  MoveL 616 to (-197.85, 161.14, -4.14) mm, rotated rx 163.15 ry -25.3 rz 35.32 deg; joints [1.714, -40.378, 129.098, -150.279, 73.685, 65.031, 129.162]
  Set speed (76.2 mm/s)
  MoveL 617 to (-197.85, 161.14, -8.4) mm, rotated rx 163.15 ry -25.3 rz 35.32 deg; joints [1.504, -40.382, 129.115, -150.492, 73.695, 65.043, 129.162]
  MoveL 618 to (-199.6, 161.14, -8.41) mm, rotated rx 163.04 ry -25.23 rz 35.58 deg; joints [1.487, -40.261, 129.125, -150.604, 73.811, 65.026, 128.915]
  MoveL 619 to (-206.05, 161.14, -11.57) mm, rotated rx 162.65 ry -24.96 rz 36.52 deg; joints [1.269, -39.819, 129.168, -151.166, 74.241, 64.973, 128.027]
  MoveL 620 to (-201.08, 161.14, -20.25) mm, rotated rx 162.95 ry -25.17 rz 35.8 deg; joints [0.888, -40.168, 129.175, -151.29, 73.933, 65.037, 128.708]
  MoveL 621 to (-201.08, 157.97, -20.25) mm, rotated rx 162.7 ry -25 rz 36.39 deg; joints [0.848, -40.277, 129.313, -151.506, 73.963, 64.865, 128.153]
  MoveL 622 to (-206.05, 157.97, -11.57) mm, rotated rx 162.4 ry -24.8 rz 37.1 deg; joints [1.229, -39.927, 129.307, -151.385, 74.271, 64.804, 127.476]
  MoveL 623 to (-199.6, 157.97, -8.41) mm, rotated rx 162.79 ry -25.06 rz 36.17 deg; joints [1.449, -40.37, 129.264, -150.819, 73.841, 64.853, 128.359]
  MoveL 624 to (-197.85, 157.97, -8.4) mm, rotated rx 162.9 ry -25.13 rz 35.91 deg; joints [1.466, -40.491, 129.254, -150.707, 73.725, 64.869, 128.605]
  MoveL 625 to (-197.85, 157.97, -4.14) mm, rotated rx 162.9 ry -25.13 rz 35.91 deg; joints [1.676, -40.487, 129.236, -150.493, 73.716, 64.858, 128.605]
  Set speed (38.1 mm/s)
  MoveL 626 to (-197.89, 157.97, -3.98) mm, rotated rx 162.9 ry -25.13 rz 35.92 deg; joints [1.684, -40.484, 129.236, -150.488, 73.718, 64.857, 128.599]
  MoveL 627 to (-198.05, 157.65, -3.7) mm, rotated rx 162.87 ry -25.11 rz 36 deg; joints [1.692, -40.484, 129.25, -150.506, 73.731, 64.838, 128.521]
  Set speed (76.2 mm/s)
  MoveL 628 to (-198.05, 155.11, -3.7) mm, rotated rx 162.66 ry -24.98 rz 36.48 deg; joints [1.661, -40.571, 129.362, -150.683, 73.756, 64.699, 128.068]
  Set speed (38.1 mm/s)
  MoveL 629 to (-197.89, 154.79, -3.98) mm, rotated rx 162.65 ry -24.97 rz 36.51 deg; joints [1.644, -40.593, 129.376, -150.709, 73.749, 64.684, 128.033]
  MoveL 630 to (-197.85, 154.79, -4.14) mm, rotated rx 162.65 ry -24.97 rz 36.51 deg; joints [1.637, -40.596, 129.377, -150.714, 73.747, 64.685, 128.039]
  Set speed (76.2 mm/s)
  MoveL 631 to (-197.85, 154.79, -8.4) mm, rotated rx 162.65 ry -24.97 rz 36.51 deg; joints [1.426, -40.6, 129.394, -150.928, 73.756, 64.695, 128.039]
  MoveL 632 to (-199.6, 154.79, -8.41) mm, rotated rx 162.54 ry -24.89 rz 36.76 deg; joints [1.409, -40.479, 129.404, -151.041, 73.873, 64.68, 127.794]
  MoveL 633 to (-206.05, 154.79, -11.57) mm, rotated rx 162.16 ry -24.63 rz 37.69 deg; joints [1.188, -40.035, 129.447, -151.609, 74.302, 64.635, 126.915]
  MoveL 634 to (-201.08, 154.79, -20.25) mm, rotated rx 162.45 ry -24.83 rz 36.98 deg; joints [0.808, -40.386, 129.453, -151.729, 73.993, 64.693, 127.59]
  MoveL 635 to (-201.08, 151.62, -20.25) mm, rotated rx 162.2 ry -24.66 rz 37.58 deg; joints [0.765, -40.493, 129.594, -151.959, 74.025, 64.521, 127.017]
  MoveL 636 to (-206.05, 151.62, -11.57) mm, rotated rx 161.91 ry -24.45 rz 38.28 deg; joints [1.146, -40.142, 129.589, -151.84, 74.333, 64.466, 126.347]
  MoveL 637 to (-199.6, 151.62, -8.41) mm, rotated rx 162.29 ry -24.72 rz 37.37 deg; joints [1.367, -40.587, 129.546, -151.27, 73.905, 64.508, 127.221]
  MoveL 638 to (-197.85, 151.62, -8.4) mm, rotated rx 162.4 ry -24.79 rz 37.11 deg; joints [1.385, -40.708, 129.536, -151.156, 73.789, 64.522, 127.465]
  MoveL 639 to (-197.85, 151.62, -4.14) mm, rotated rx 162.4 ry -24.79 rz 37.11 deg; joints [1.596, -40.704, 129.519, -150.942, 73.779, 64.512, 127.465]
  Set speed (38.1 mm/s)
  MoveL 640 to (-197.89, 151.62, -3.98) mm, rotated rx 162.39 ry -24.79 rz 37.12 deg; joints [1.604, -40.701, 129.518, -150.937, 73.782, 64.511, 127.459]
  MoveL 641 to (-198.05, 151.3, -3.7) mm, rotated rx 162.36 ry -24.77 rz 37.2 deg; joints [1.612, -40.701, 129.533, -150.956, 73.795, 64.492, 127.378]
  Set speed (76.2 mm/s)
  MoveL 642 to (-198.05, 148.76, -3.7) mm, rotated rx 162.15 ry -24.63 rz 37.69 deg; joints [1.578, -40.786, 129.648, -151.144, 73.821, 64.354, 126.912]
  Set speed (38.1 mm/s)
  MoveL 643 to (-197.89, 148.44, -3.98) mm, rotated rx 162.14 ry -24.62 rz 37.73 deg; joints [1.562, -40.808, 129.663, -151.171, 73.815, 64.339, 126.875]
  MoveL 644 to (-197.85, 148.44, -4.14) mm, rotated rx 162.14 ry -24.62 rz 37.72 deg; joints [1.554, -40.812, 129.663, -151.176, 73.812, 64.339, 126.881]
  Set speed (76.2 mm/s)
  MoveL 645 to (-197.85, 148.44, -8.4) mm, rotated rx 162.14 ry -24.62 rz 37.72 deg; joints [1.343, -40.815, 129.68, -151.391, 73.822, 64.35, 126.881]
  MoveL 646 to (-199.6, 148.44, -8.41) mm, rotated rx 162.04 ry -24.54 rz 37.98 deg; joints [1.325, -40.694, 129.69, -151.505, 73.937, 64.337, 126.639]
  MoveL 647 to (-206.05, 148.44, -11.57) mm, rotated rx 161.66 ry -24.27 rz 38.88 deg; joints [1.102, -40.248, 129.733, -152.077, 74.366, 64.298, 125.77]
  MoveL 648 to (-201.08, 148.44, -20.25) mm, rotated rx 161.95 ry -24.48 rz 38.19 deg; joints [0.722, -40.6, 129.738, -152.196, 74.058, 64.349, 126.436]
  MoveL 649 to (-201.08, 145.27, -20.25) mm, rotated rx 161.69 ry -24.3 rz 38.8 deg; joints [0.676, -40.706, 129.883, -152.439, 74.091, 64.178, 125.846]
  MoveL 650 to (-206.05, 145.27, -11.57) mm, rotated rx 161.41 ry -24.09 rz 39.49 deg; joints [1.057, -40.353, 129.879, -152.322, 74.399, 64.131, 125.185]
  MoveL 651 to (-199.6, 145.27, -8.41) mm, rotated rx 161.78 ry -24.36 rz 38.59 deg; joints [1.28, -40.8, 129.836, -151.748, 73.971, 64.166, 126.047]
  MoveL 652 to (-197.85, 145.27, -8.4) mm, rotated rx 161.88 ry -24.43 rz 38.34 deg; joints [1.299, -40.922, 129.826, -151.633, 73.856, 64.178, 126.288]
  MoveL 653 to (-197.85, 145.27, -4.14) mm, rotated rx 161.88 ry -24.43 rz 38.34 deg; joints [1.51, -40.918, 129.809, -151.418, 73.846, 64.168, 126.288]
  Set speed (38.1 mm/s)
  MoveL 654 to (-197.89, 145.27, -3.98) mm, rotated rx 161.88 ry -24.43 rz 38.35 deg; joints [1.518, -40.915, 129.809, -151.413, 73.849, 64.167, 126.282]
  MoveL 655 to (-198.05, 144.95, -3.7) mm, rotated rx 161.85 ry -24.41 rz 38.43 deg; joints [1.525, -40.914, 129.824, -151.434, 73.862, 64.148, 126.2]
  Set speed (76.2 mm/s)
  MoveL 656 to (-198.05, 142.41, -3.7) mm, rotated rx 161.64 ry -24.26 rz 38.94 deg; joints [1.489, -40.999, 129.942, -151.633, 73.89, 64.011, 125.719]
  Set speed (38.1 mm/s)
  MoveL 657 to (-197.89, 142.09, -3.98) mm, rotated rx 161.62 ry -24.24 rz 38.98 deg; joints [1.473, -41.021, 129.957, -151.662, 73.884, 63.996, 125.68]
  MoveL 658 to (-197.85, 142.09, -4.14) mm, rotated rx 161.62 ry -24.25 rz 38.97 deg; joints [1.465, -41.024, 129.958, -151.667, 73.881, 63.996, 125.686]
  Set speed (76.2 mm/s)
  MoveL 659 to (-197.85, 142.09, -8.4) mm, rotated rx 161.62 ry -24.25 rz 38.97 deg; joints [1.253, -41.028, 129.974, -151.882, 73.89, 64.006, 125.686]
  MoveL 660 to (-199.6, 142.09, -8.41) mm, rotated rx 161.52 ry -24.17 rz 39.22 deg; joints [1.235, -40.905, 129.984, -151.997, 74.006, 63.995, 125.447]
  MoveL 661 to (-206.05, 142.09, -11.57) mm, rotated rx 161.16 ry -23.9 rz 40.11 deg; joints [1.01, -40.458, 130.027, -152.573, 74.433, 63.964, 124.591]
  MoveL 662 to (-201.08, 142.09, -20.25) mm, rotated rx 161.44 ry -24.11 rz 39.43 deg; joints [0.63, -40.811, 130.03, -152.69, 74.125, 64.008, 125.247]
  MoveL 663 to (-201.08, 138.92, -20.25) mm, rotated rx 161.18 ry -23.91 rz 40.06 deg; joints [0.581, -40.915, 130.18, -152.948, 74.16, 63.838, 124.639]
  MoveL 664 to (-206.05, 138.92, -11.57) mm, rotated rx 160.91 ry -23.7 rz 40.73 deg; joints [0.962, -40.561, 130.176, -152.831, 74.467, 63.797, 123.988]
  MoveL 665 to (-199.6, 138.92, -8.41) mm, rotated rx 161.26 ry -23.98 rz 39.85 deg; joints [1.187, -41.01, 130.134, -152.254, 74.041, 63.825, 124.838]
  MoveL 666 to (-197.85, 138.92, -8.4) mm, rotated rx 161.37 ry -24.05 rz 39.6 deg; joints [1.206, -41.133, 130.124, -152.138, 73.926, 63.835, 125.075]
  MoveL 667 to (-197.85, 138.92, -4.14) mm, rotated rx 161.37 ry -24.05 rz 39.6 deg; joints [1.418, -41.129, 130.108, -151.923, 73.917, 63.826, 125.075]
  Set speed (38.1 mm/s)
  MoveL 668 to (-197.89, 138.92, -3.98) mm, rotated rx 161.36 ry -24.05 rz 39.61 deg; joints [1.426, -41.126, 130.108, -151.918, 73.919, 63.825, 125.069]
  MoveL 669 to (-198.05, 138.6, -3.7) mm, rotated rx 161.33 ry -24.02 rz 39.7 deg; joints [1.433, -41.125, 130.123, -151.941, 73.932, 63.806, 124.986]
  Set speed (76.2 mm/s)
  MoveL 670 to (-198.05, 136.06, -3.7) mm, rotated rx 161.12 ry -23.86 rz 40.21 deg; joints [1.394, -41.209, 130.245, -152.152, 73.961, 63.671, 124.49]
  Set speed (38.1 mm/s)
  MoveL 671 to (-197.89, 135.74, -3.98) mm, rotated rx 161.1 ry -23.85 rz 40.25 deg; joints [1.378, -41.23, 130.26, -152.182, 73.955, 63.655, 124.449]
  MoveL 672 to (-197.85, 135.74, -4.14) mm, rotated rx 161.1 ry -23.85 rz 40.25 deg; joints [1.37, -41.234, 130.26, -152.187, 73.953, 63.656, 124.454]
  Set speed (76.2 mm/s)
  MoveL 673 to (-197.85, 135.74, -8.4) mm, rotated rx 161.1 ry -23.85 rz 40.25 deg; joints [1.158, -41.237, 130.276, -152.402, 73.962, 63.665, 124.454]
  MoveL 674 to (-199.6, 135.74, -8.41) mm, rotated rx 161.01 ry -23.78 rz 40.49 deg; joints [1.138, -41.114, 130.286, -152.519, 74.077, 63.656, 124.219]
  MoveL 675 to (-206.05, 135.74, -11.57) mm, rotated rx 160.66 ry -23.5 rz 41.36 deg; joints [0.913, -40.665, 130.328, -153.097, 74.502, 63.632, 123.377]
  MoveL 676 to (-201.08, 135.74, -20.25) mm, rotated rx 160.92 ry -23.71 rz 40.69 deg; joints [0.531, -41.019, 130.331, -153.213, 74.196, 63.669, 124.023]
  MoveL 677 to (-201.08, 132.57, -20.25) mm, rotated rx 160.67 ry -23.51 rz 41.34 deg; joints [0.48, -41.122, 130.484, -153.485, 74.232, 63.5, 123.397]
  MoveL 678 to (-206.05, 132.57, -11.57) mm, rotated rx 160.4 ry -23.29 rz 42 deg; joints [0.861, -40.767, 130.481, -153.369, 74.538, 63.467, 122.757]
  MoveL 679 to (-199.6, 132.57, -8.41) mm, rotated rx 160.75 ry -23.57 rz 41.14 deg; joints [1.088, -41.218, 130.44, -152.79, 74.113, 63.487, 123.591]
  MoveL 680 to (-197.85, 132.57, -8.4) mm, rotated rx 160.84 ry -23.65 rz 40.9 deg; joints [1.107, -41.341, 130.43, -152.674, 73.999, 63.495, 123.825]
  MoveL 681 to (-197.85, 132.57, -4.14) mm, rotated rx 160.84 ry -23.65 rz 40.9 deg; joints [1.32, -41.337, 130.415, -152.458, 73.99, 63.486, 123.825]
  Set speed (38.1 mm/s)
  MoveL 682 to (-197.89, 132.57, -3.98) mm, rotated rx 160.84 ry -23.64 rz 40.9 deg; joints [1.328, -41.334, 130.415, -152.453, 73.992, 63.486, 123.819]
  MoveL 683 to (-198.05, 132.25, -3.7) mm, rotated rx 160.8 ry -23.62 rz 40.99 deg; joints [1.334, -41.333, 130.43, -152.478, 74.006, 63.468, 123.734]
  Set speed (76.2 mm/s)
  MoveL 684 to (-198.05, 129.71, -3.7) mm, rotated rx 160.59 ry -23.45 rz 41.52 deg; joints [1.293, -41.416, 130.555, -152.701, 74.036, 63.333, 123.223]
  Set speed (38.1 mm/s)
  MoveL 685 to (-197.89, 129.39, -3.98) mm, rotated rx 160.58 ry -23.43 rz 41.56 deg; joints [1.276, -41.437, 130.571, -152.732, 74.029, 63.318, 123.18]
  MoveL 686 to (-197.85, 129.39, -4.14) mm, rotated rx 160.58 ry -23.44 rz 41.56 deg; joints [1.268, -41.441, 130.572, -152.738, 74.027, 63.318, 123.185]
  Set speed (76.2 mm/s)
  MoveL 687 to (-197.85, 129.39, -8.4) mm, rotated rx 160.58 ry -23.44 rz 41.56 deg; joints [1.055, -41.444, 130.587, -152.953, 74.036, 63.327, 123.185]
  MoveL 688 to (-199.6, 129.39, -8.41) mm, rotated rx 160.49 ry -23.36 rz 41.79 deg; joints [1.036, -41.321, 130.597, -153.07, 74.15, 63.32, 122.954]
  MoveL 689 to (-206.05, 129.39, -11.57) mm, rotated rx 160.15 ry -23.08 rz 42.64 deg; joints [0.808, -40.869, 130.637, -153.649, 74.574, 63.303, 122.128]
  MoveL 690 to (-201.08, 129.39, -20.25) mm, rotated rx 160.41 ry -23.29 rz 41.99 deg; joints [0.426, -41.225, 130.639, -153.766, 74.268, 63.333, 122.761]
  MoveL 691 to (-201.08, 126.22, -20.25) mm, rotated rx 160.15 ry -23.08 rz 42.65 deg; joints [0.371, -41.327, 130.797, -154.054, 74.305, 63.166, 122.117]
  MoveL 692 to (-206.05, 126.22, -11.57) mm, rotated rx 159.9 ry -22.86 rz 43.29 deg; joints [0.753, -40.97, 130.794, -153.937, 74.61, 63.14, 121.49]
  MoveL 693 to (-199.6, 126.22, -8.41) mm, rotated rx 160.22 ry -23.14 rz 42.46 deg; joints [0.982, -41.423, 130.755, -153.357, 74.188, 63.153, 122.308]
  MoveL 694 to (-197.85, 126.22, -8.4) mm, rotated rx 160.32 ry -23.22 rz 42.22 deg; joints [1.001, -41.546, 130.745, -153.24, 74.074, 63.159, 122.537]
  MoveL 695 to (-197.85, 126.22, -4.14) mm, rotated rx 160.32 ry -23.22 rz 42.22 deg; joints [1.215, -41.543, 130.73, -153.025, 74.065, 63.151, 122.537]
  Set speed (38.1 mm/s)
  MoveL 696 to (-197.89, 126.22, -3.98) mm, rotated rx 160.31 ry -23.22 rz 42.23 deg; joints [1.222, -41.54, 130.73, -153.019, 74.067, 63.15, 122.531]
  MoveL 697 to (-198.05, 125.9, -3.7) mm, rotated rx 160.28 ry -23.19 rz 42.32 deg; joints [1.229, -41.539, 130.746, -153.045, 74.081, 63.133, 122.445]
  Set speed (76.2 mm/s)
  MoveL 698 to (-198.05, 123.36, -3.7) mm, rotated rx 160.07 ry -23.01 rz 42.85 deg; joints [1.185, -41.62, 130.875, -153.281, 74.112, 63, 121.919]
  Set speed (38.1 mm/s)
  MoveL 699 to (-197.89, 123.04, -3.98) mm, rotated rx 160.05 ry -22.99 rz 42.9 deg; joints [1.167, -41.642, 130.891, -153.314, 74.106, 62.984, 121.873]
  MoveL 700 to (-197.85, 123.04, -4.14) mm, rotated rx 160.05 ry -23 rz 42.9 deg; joints [1.16, -41.645, 130.891, -153.32, 74.103, 62.984, 121.879]
  Set speed (76.2 mm/s)
  MoveL 701 to (-197.85, 123.04, -8.4) mm, rotated rx 160.05 ry -23 rz 42.9 deg; joints [0.946, -41.648, 130.906, -153.536, 74.112, 62.992, 121.879]
  MoveL 702 to (-199.6, 123.04, -8.41) mm, rotated rx 159.96 ry -22.92 rz 43.13 deg; joints [0.926, -41.525, 130.915, -153.653, 74.226, 62.988, 121.652]
  MoveL 703 to (-206.05, 123.04, -11.57) mm, rotated rx 159.64 ry -22.64 rz 43.95 deg; joints [0.697, -41.071, 130.953, -154.231, 74.647, 62.978, 120.844]
  MoveL 704 to (-201.08, 123.04, -20.25) mm, rotated rx 159.89 ry -22.85 rz 43.32 deg; joints [0.315, -41.428, 130.956, -154.35, 74.343, 63.001, 121.464]
  MoveL 705 to (-201.08, 119.87, -20.25) mm, rotated rx 159.63 ry -22.62 rz 43.99 deg; joints [0.256, -41.529, 131.117, -154.654, 74.38, 62.836, 120.801]
  MoveL 706 to (-206.05, 119.87, -11.57) mm, rotated rx 159.39 ry -22.41 rz 44.61 deg; joints [0.639, -41.171, 131.114, -154.534, 74.684, 62.817, 120.189]
  MoveL 707 to (-199.6, 119.87, -8.41) mm, rotated rx 159.7 ry -22.69 rz 43.8 deg; joints [0.868, -41.626, 131.078, -153.956, 74.264, 62.823, 120.987]
  MoveL 708 to (-197.85, 119.87, -8.4) mm, rotated rx 159.79 ry -22.77 rz 43.58 deg; joints [0.888, -41.75, 131.068, -153.839, 74.15, 62.827, 121.211]
  MoveL 709 to (-197.85, 119.87, -4.14) mm, rotated rx 159.79 ry -22.77 rz 43.58 deg; joints [1.103, -41.747, 131.054, -153.623, 74.142, 62.819, 121.211]
  Set speed (38.1 mm/s)
  MoveL 710 to (-197.89, 119.87, -3.98) mm, rotated rx 159.78 ry -22.76 rz 43.58 deg; joints [1.11, -41.744, 131.054, -153.618, 74.144, 62.819, 121.205]
  MoveL 711 to (-198.05, 119.55, -3.7) mm, rotated rx 159.75 ry -22.73 rz 43.67 deg; joints [1.116, -41.742, 131.07, -153.645, 74.158, 62.802, 121.118]
  Set speed (76.2 mm/s)
  MoveL 712 to (-198.05, 117.01, -3.7) mm, rotated rx 159.54 ry -22.55 rz 44.22 deg; joints [1.069, -41.823, 131.203, -153.894, 74.189, 62.671, 120.576]
  Set speed (38.1 mm/s)
  MoveL 713 to (-197.89, 116.7, -3.98) mm, rotated rx 159.52 ry -22.53 rz 44.27 deg; joints [1.051, -41.845, 131.219, -153.929, 74.183, 62.655, 120.528]
  MoveL 714 to (-197.85, 116.7, -4.14) mm, rotated rx 159.52 ry -22.53 rz 44.26 deg; joints [1.044, -41.848, 131.22, -153.934, 74.181, 62.655, 120.533]
  Set speed (76.2 mm/s)
  MoveL 715 to (-197.85, 116.7, -8.4) mm, rotated rx 159.52 ry -22.53 rz 44.26 deg; joints [0.829, -41.851, 131.233, -154.151, 74.189, 62.662, 120.533]
  MoveL 716 to (-199.6, 116.7, -8.41) mm, rotated rx 159.44 ry -22.45 rz 44.49 deg; joints [0.809, -41.727, 131.242, -154.267, 74.302, 62.66, 120.313]
  MoveL 717 to (-206.05, 116.7, -11.57) mm, rotated rx 159.13 ry -22.17 rz 45.28 deg; joints [0.579, -41.271, 131.277, -154.845, 74.721, 62.657, 119.525]
  MoveL 718 to (-201.08, 116.7, -20.25) mm, rotated rx 159.37 ry -22.39 rz 44.67 deg; joints [0.195, -41.629, 131.28, -154.965, 74.418, 62.672, 120.129]
  MoveL 719 to (-201.08, 113.52, -20.25) mm, rotated rx 159.1 ry -22.15 rz 45.36 deg; joints [0.133, -41.729, 131.446, -155.286, 74.456, 62.51, 119.447]
  MoveL 720 to (-206.05, 113.52, -11.57) mm, rotated rx 158.88 ry -21.93 rz 45.96 deg; joints [0.517, -41.37, 131.442, -155.163, 74.758, 62.499, 118.852]
  MoveL 721 to (-199.6, 113.52, -8.41) mm, rotated rx 159.17 ry -22.21 rz 45.18 deg; joints [0.748, -41.827, 131.409, -154.587, 74.341, 62.498, 119.629]
  MoveL 722 to (-197.85, 113.52, -8.4) mm, rotated rx 159.26 ry -22.29 rz 44.96 deg; joints [0.768, -41.951, 131.4, -154.471, 74.228, 62.499, 119.847]
  MoveL 723 to (-197.85, 113.52, -4.14) mm, rotated rx 159.26 ry -22.29 rz 44.96 deg; joints [0.983, -41.948, 131.387, -154.254, 74.22, 62.492, 119.847]
  Set speed (38.1 mm/s)
  MoveL 724 to (-197.89, 113.52, -3.98) mm, rotated rx 159.25 ry -22.29 rz 44.96 deg; joints [0.99, -41.945, 131.387, -154.249, 74.222, 62.492, 119.841]
  MoveL 725 to (-198.05, 113.2, -3.7) mm, rotated rx 159.22 ry -22.26 rz 45.05 deg; joints [0.996, -41.944, 131.403, -154.278, 74.236, 62.475, 119.752]
  Set speed (76.2 mm/s)
  MoveL 726 to (-198.05, 110.66, -3.7) mm, rotated rx 159.01 ry -22.06 rz 45.62 deg; joints [0.946, -42.024, 131.539, -154.541, 74.267, 62.347, 119.195]
  Set speed (38.1 mm/s)
  MoveL 727 to (-197.89, 110.35, -3.98) mm, rotated rx 158.99 ry -22.04 rz 45.67 deg; joints [0.927, -42.045, 131.556, -154.577, 74.261, 62.331, 119.145]
  MoveL 728 to (-197.85, 110.35, -4.14) mm, rotated rx 158.99 ry -22.04 rz 45.66 deg; joints [0.92, -42.048, 131.556, -154.583, 74.259, 62.331, 119.15]
  Set speed (76.2 mm/s)
  MoveL 729 to (-197.85, 110.35, -8.4) mm, rotated rx 158.99 ry -22.04 rz 45.66 deg; joints [0.704, -42.051, 131.57, -154.8, 74.267, 62.337, 119.15]
  MoveL 730 to (-199.6, 110.35, -8.41) mm, rotated rx 158.91 ry -21.96 rz 45.88 deg; joints [0.684, -41.927, 131.578, -154.915, 74.38, 62.337, 118.936]
  MoveL 731 to (-206.05, 110.35, -11.57) mm, rotated rx 158.63 ry -21.69 rz 46.65 deg; joints [0.453, -41.469, 131.609, -155.489, 74.795, 62.342, 118.171]
  MoveL 732 to (-201.08, 110.35, -20.25) mm, rotated rx 158.84 ry -21.9 rz 46.06 deg; joints [0.068, -41.828, 131.613, -155.614, 74.494, 62.349, 118.757]
  MoveL 733 to (-201.08, 107.17, -20.25) mm, rotated rx 158.58 ry -21.64 rz 46.76 deg; joints [0.002, -41.927, 131.782, -155.951, 74.532, 62.19, 118.057]
  MoveL 734 to (-206.05, 107.17, -11.57) mm, rotated rx 158.37 ry -21.43 rz 47.34 deg; joints [0.387, -41.567, 131.777, -155.823, 74.832, 62.186, 117.48]
  MoveL 735 to (-199.6, 107.17, -8.41) mm, rotated rx 158.65 ry -21.71 rz 46.58 deg; joints [0.619, -42.026, 131.748, -155.252, 74.418, 62.178, 118.233]
  MoveL 736 to (-197.85, 107.17, -8.4) mm, rotated rx 158.73 ry -21.79 rz 46.37 deg; joints [0.639, -42.151, 131.741, -155.137, 74.306, 62.177, 118.444]
  MoveL 737 to (-197.85, 107.17, -4.14) mm, rotated rx 158.73 ry -21.79 rz 46.37 deg; joints [0.855, -42.148, 131.728, -154.919, 74.298, 62.171, 118.444]
  Set speed (38.1 mm/s)
  MoveL 738 to (-197.89, 107.17, -3.98) mm, rotated rx 158.72 ry -21.78 rz 46.38 deg; joints [0.862, -42.145, 131.728, -154.914, 74.3, 62.171, 118.439]
  MoveL 739 to (-198.05, 106.85, -3.7) mm, rotated rx 158.69 ry -21.75 rz 46.47 deg; joints [0.868, -42.143, 131.745, -154.945, 74.314, 62.155, 118.348]
  Set speed (76.2 mm/s)
  MoveL 740 to (-198.05, 104.31, -3.7) mm, rotated rx 158.48 ry -21.54 rz 47.04 deg; joints [0.814, -42.223, 131.884, -155.221, 74.345, 62.029, 117.776]
  Set speed (38.1 mm/s)
  MoveL 741 to (-197.89, 104, -3.98) mm, rotated rx 158.46 ry -21.52 rz 47.09 deg; joints [0.795, -42.244, 131.902, -155.26, 74.339, 62.013, 117.723]
  MoveL 742 to (-197.85, 104, -4.14) mm, rotated rx 158.46 ry -21.52 rz 47.09 deg; joints [0.788, -42.247, 131.902, -155.265, 74.337, 62.013, 117.728]
  Set speed (76.2 mm/s)
  MoveL 743 to (-197.85, 104, -8.4) mm, rotated rx 158.46 ry -21.52 rz 47.09 deg; joints [0.572, -42.25, 131.914, -155.483, 74.345, 62.018, 117.728]
  MoveL 744 to (-199.6, 104, -8.41) mm, rotated rx 158.39 ry -21.45 rz 47.3 deg; joints [0.551, -42.125, 131.921, -155.597, 74.456, 62.021, 117.521]
  MoveL 745 to (-206.05, 104, -11.57) mm, rotated rx 158.12 ry -21.17 rz 48.03 deg; joints [0.319, -41.665, 131.947, -156.166, 74.869, 62.032, 116.781]
  MoveL 746 to (-201.08, 104, -20.25) mm, rotated rx 158.32 ry -21.38 rz 47.47 deg; joints [-0.067, -42.025, 131.954, -156.296, 74.569, 62.032, 117.348]
  MoveL 747 to (-201.08, 100.82, -20.25) mm, rotated rx 158.06 ry -21.12 rz 48.18 deg; joints [-0.137, -42.123, 132.127, -156.65, 74.606, 61.876, 116.63]
  MoveL 748 to (-206.05, 100.82, -11.57) mm, rotated rx 157.87 ry -20.91 rz 48.74 deg; joints [0.25, -41.762, 132.12, -156.516, 74.905, 61.88, 116.073]
  MoveL 749 to (-199.6, 100.82, -8.41) mm, rotated rx 158.12 ry -21.18 rz 48.02 deg; joints [0.482, -42.223, 132.096, -155.951, 74.495, 61.865, 116.799]
  MoveL 750 to (-197.85, 100.82, -8.4) mm, rotated rx 158.2 ry -21.26 rz 47.81 deg; joints [0.502, -42.349, 132.09, -155.837, 74.383, 61.862, 117.003]
  MoveL 751 to (-197.85, 100.82, -4.14) mm, rotated rx 158.2 ry -21.26 rz 47.81 deg; joints [0.719, -42.346, 132.078, -155.619, 74.375, 61.857, 117.003]
  Set speed (38.1 mm/s)
  MoveL 752 to (-197.89, 100.82, -3.98) mm, rotated rx 158.2 ry -21.25 rz 47.82 deg; joints [0.726, -42.343, 132.077, -155.614, 74.378, 61.857, 116.998]
  MoveL 753 to (-198.05, 100.5, -3.7) mm, rotated rx 158.16 ry -21.22 rz 47.91 deg; joints [0.731, -42.341, 132.095, -155.646, 74.391, 61.841, 116.907]
  Set speed (76.2 mm/s)
  MoveL 754 to (-198.05, 97.96, -3.7) mm, rotated rx 157.95 ry -21 rz 48.49 deg; joints [0.674, -42.42, 132.237, -155.937, 74.422, 61.717, 116.319]
  Set speed (38.1 mm/s)
  MoveL 755 to (-197.89, 97.65, -3.98) mm, rotated rx 157.93 ry -20.98 rz 48.55 deg; joints [0.655, -42.442, 132.255, -155.977, 74.416, 61.702, 116.264]
  MoveL 756 to (-197.85, 97.65, -4.14) mm, rotated rx 157.93 ry -20.98 rz 48.54 deg; joints [0.647, -42.445, 132.255, -155.982, 74.414, 61.702, 116.269]
  Set speed (76.2 mm/s)
  MoveL 757 to (-197.85, 97.65, -8.4) mm, rotated rx 157.93 ry -20.98 rz 48.54 deg; joints [0.43, -42.447, 132.267, -156.201, 74.421, 61.706, 116.269]
  MoveL 758 to (-199.6, 97.65, -8.41) mm, rotated rx 157.86 ry -20.91 rz 48.74 deg; joints [0.41, -42.322, 132.273, -156.313, 74.532, 61.711, 116.069]
  MoveL 759 to (-206.05, 97.65, -11.57) mm, rotated rx 157.61 ry -20.64 rz 49.45 deg; joints [0.178, -41.859, 132.294, -156.875, 74.941, 61.73, 115.356]
  MoveL 760 to (-201.08, 97.65, -20.25) mm, rotated rx 157.81 ry -20.84 rz 48.91 deg; joints [-0.21, -42.221, 132.302, -157.012, 74.643, 61.722, 115.902]
  MoveL 761 to (-201.08, 94.47, -20.25) mm, rotated rx 157.55 ry -20.56 rz 49.63 deg; joints [-0.285, -42.318, 132.479, -157.383, 74.68, 61.569, 115.166]
  MoveL 762 to (-206.05, 94.47, -11.57) mm, rotated rx 157.36 ry -20.36 rz 50.16 deg; joints [0.104, -41.955, 132.469, -157.242, 74.977, 61.581, 114.631]
  MoveL 763 to (-199.6, 94.47, -8.41) mm, rotated rx 157.6 ry -20.63 rz 49.47 deg; joints [0.336, -42.419, 132.451, -156.684, 74.569, 61.559, 115.329]
  MoveL 764 to (-197.85, 94.47, -8.4) mm, rotated rx 157.67 ry -20.7 rz 49.28 deg; joints [0.357, -42.546, 132.446, -156.573, 74.459, 61.553, 115.525]
  MoveL 765 to (-197.85, 94.47, -4.14) mm, rotated rx 157.67 ry -20.7 rz 49.28 deg; joints [0.574, -42.543, 132.435, -156.354, 74.451, 61.549, 115.525]
  Set speed (38.1 mm/s)
  MoveL 766 to (-197.89, 94.47, -3.98) mm, rotated rx 157.67 ry -20.7 rz 49.28 deg; joints [0.582, -42.54, 132.435, -156.349, 74.454, 61.549, 115.52]
  MoveL 767 to (-198.05, 94.15, -3.7) mm, rotated rx 157.64 ry -20.66 rz 49.38 deg; joints [0.586, -42.538, 132.453, -156.383, 74.467, 61.534, 115.427]
  Set speed (76.2 mm/s)
  MoveL 768 to (-198.05, 91.61, -3.7) mm, rotated rx 157.43 ry -20.43 rz 49.97 deg; joints [0.526, -42.617, 132.598, -156.687, 74.497, 61.414, 114.825]
  Set speed (38.1 mm/s)
  MoveL 769 to (-197.89, 91.3, -3.98) mm, rotated rx 157.41 ry -20.41 rz 50.03 deg; joints [0.506, -42.638, 132.617, -156.73, 74.491, 61.399, 114.767]
  MoveL 770 to (-197.85, 91.3, -4.14) mm, rotated rx 157.41 ry -20.41 rz 50.02 deg; joints [0.498, -42.641, 132.617, -156.735, 74.489, 61.399, 114.771]
  Set speed (76.2 mm/s)
  MoveL 771 to (-197.85, 91.3, -8.4) mm, rotated rx 157.41 ry -20.41 rz 50.02 deg; joints [0.28, -42.644, 132.628, -156.954, 74.496, 61.402, 114.771]
  MoveL 772 to (-200.08, 91.3, -8.41) mm, rotated rx 157.33 ry -20.32 rz 50.26 deg; joints [0.255, -42.482, 132.633, -157.094, 74.636, 61.41, 114.527]
  MoveL 773 to (-206.05, 91.3, -11.57) mm, rotated rx 157.11 ry -20.08 rz 50.88 deg; joints [0.028, -42.052, 132.647, -157.617, 75.012, 61.434, 113.897]
  MoveL 774 to (-201.08, 91.3, -20.25) mm, rotated rx 157.29 ry -20.28 rz 50.37 deg; joints [-0.362, -42.415, 132.657, -157.763, 74.716, 61.419, 114.42]
  MoveL 775 to (-201.08, 88.12, -20.25) mm, rotated rx 157.04 ry -19.99 rz 51.11 deg; joints [-0.441, -42.512, 132.838, -158.151, 74.751, 61.27, 113.666]
  MoveL 776 to (-206.05, 88.12, -11.57) mm, rotated rx 156.87 ry -19.79 rz 51.61 deg; joints [-0.05, -42.147, 132.826, -158.001, 75.046, 61.29, 113.155]
  MoveL 777 to (-200.08, 88.12, -8.41) mm, rotated rx 157.07 ry -20.03 rz 51.01 deg; joints [0.177, -42.579, 132.815, -157.483, 74.672, 61.263, 113.77]
  MoveL 778 to (-197.85, 88.12, -8.4) mm, rotated rx 157.15 ry -20.12 rz 50.77 deg; joints [0.202, -42.741, 132.811, -157.344, 74.533, 61.253, 114.009]
  MoveL 779 to (-197.85, 88.12, -4.14) mm, rotated rx 157.15 ry -20.12 rz 50.77 deg; joints [0.42, -42.739, 132.801, -157.125, 74.525, 61.25, 114.009]
  Set speed (38.1 mm/s)
  MoveL 780 to (-197.89, 88.12, -3.98) mm, rotated rx 157.15 ry -20.12 rz 50.78 deg; joints [0.428, -42.736, 132.8, -157.12, 74.528, 61.25, 114.004]
  MoveL 781 to (-198.05, 87.81, -3.7) mm, rotated rx 157.12 ry -20.08 rz 50.87 deg; joints [0.432, -42.734, 132.818, -157.155, 74.541, 61.236, 113.91]
  Set speed (76.2 mm/s)
  MoveL 782 to (-198.05, 85.27, -3.7) mm, rotated rx 156.91 ry -19.84 rz 51.47 deg; joints [0.368, -42.812, 132.967, -157.474, 74.569, 61.119, 113.293]
  Set speed (38.1 mm/s)
  MoveL 783 to (-197.89, 84.95, -3.98) mm, rotated rx 156.89 ry -19.82 rz 51.53 deg; joints [0.348, -42.833, 132.986, -157.519, 74.563, 61.104, 113.233]
  MoveL 784 to (-197.85, 84.95, -4.14) mm, rotated rx 156.89 ry -19.82 rz 51.53 deg; joints [0.34, -42.837, 132.986, -157.524, 74.561, 61.104, 113.237]
  Set speed (76.2 mm/s)
  MoveL 785 to (-197.85, 84.95, -8.4) mm, rotated rx 156.89 ry -19.82 rz 51.53 deg; joints [0.121, -42.839, 132.996, -157.744, 74.568, 61.107, 113.237]
  MoveL 786 to (-200.08, 84.95, -8.41) mm, rotated rx 156.82 ry -19.73 rz 51.76 deg; joints [0.096, -42.676, 132.999, -157.88, 74.707, 61.117, 113.004]
  MoveL 787 to (-206.05, 84.95, -11.57) mm, rotated rx 156.62 ry -19.49 rz 52.34 deg; joints [-0.13, -42.243, 133.006, -158.393, 75.08, 61.147, 112.405]
  MoveL 788 to (-201.08, 84.95, -20.25) mm, rotated rx 156.78 ry -19.69 rz 51.86 deg; joints [-0.523, -42.609, 133.02, -158.548, 74.785, 61.124, 112.902]
  MoveL 789 to (-201.08, 81.77, -20.25) mm, rotated rx 156.53 ry -19.38 rz 52.61 deg; joints [-0.607, -42.705, 133.204, -158.954, 74.818, 60.98, 112.13]
  MoveL 790 to (-206.05, 81.77, -11.57) mm, rotated rx 156.38 ry -19.19 rz 53.08 deg; joints [-0.213, -42.338, 133.188, -158.793, 75.112, 61.007, 111.646]
  MoveL 791 to (-200.08, 81.77, -8.41) mm, rotated rx 156.56 ry -19.42 rz 52.51 deg; joints [0.014, -42.773, 133.184, -158.286, 74.741, 60.975, 112.23]
  MoveL 792 to (-197.85, 81.77, -8.4) mm, rotated rx 156.64 ry -19.51 rz 52.29 deg; joints [0.038, -42.936, 133.183, -158.152, 74.603, 60.962, 112.456]
  MoveL 793 to (-197.85, 81.77, -4.14) mm, rotated rx 156.64 ry -19.51 rz 52.29 deg; joints [0.258, -42.934, 133.173, -157.932, 74.596, 60.961, 112.456]
  Set speed (38.1 mm/s)
  MoveL 794 to (-197.89, 81.77, -3.98) mm, rotated rx 156.64 ry -19.51 rz 52.3 deg; joints [0.265, -42.931, 133.173, -157.927, 74.598, 60.961, 112.452]
  MoveL 795 to (-198.05, 81.46, -3.7) mm, rotated rx 156.61 ry -19.47 rz 52.39 deg; joints [0.269, -42.929, 133.191, -157.963, 74.611, 60.947, 112.357]
  Set speed (76.2 mm/s)
  MoveL 796 to (-198.05, 78.92, -3.7) mm, rotated rx 156.4 ry -19.22 rz 53 deg; joints [0.202, -43.006, 133.342, -158.297, 74.638, 60.835, 111.726]
  Set speed (38.1 mm/s)
  MoveL 797 to (-197.89, 78.6, -3.98) mm, rotated rx 156.38 ry -19.19 rz 53.06 deg; joints [0.181, -43.028, 133.362, -158.343, 74.632, 60.82, 111.662]
  MoveL 798 to (-197.85, 78.6, -4.14) mm, rotated rx 156.38 ry -19.19 rz 53.06 deg; joints [0.173, -43.031, 133.362, -158.349, 74.629, 60.82, 111.667]
  Set speed (76.2 mm/s)
  MoveL 799 to (-197.85, 78.6, -8.4) mm, rotated rx 156.38 ry -19.19 rz 53.06 deg; joints [-0.047, -43.033, 133.371, -158.569, 74.636, 60.821, 111.667]
  MoveL 800 to (-200.08, 78.6, -8.41) mm, rotated rx 156.31 ry -19.11 rz 53.27 deg; joints [-0.071, -42.87, 133.371, -158.701, 74.774, 60.834, 111.446]
  MoveL 801 to (-206.05, 78.6, -11.57) mm, rotated rx 156.13 ry -18.88 rz 53.82 deg; joints [-0.297, -42.433, 133.371, -159.201, 75.144, 60.87, 110.88]
  MoveL 802 to (-201.08, 78.6, -20.25) mm, rotated rx 156.28 ry -19.07 rz 53.37 deg; joints [-0.693, -42.801, 133.389, -159.369, 74.85, 60.839, 111.35]
  MoveL 803 to (-201.08, 75.42, -20.25) mm, rotated rx 156.04 ry -18.75 rz 54.13 deg; joints [-0.782, -42.897, 133.575, -159.792, 74.881, 60.701, 110.561]
  MoveL 804 to (-206.05, 75.42, -11.57) mm, rotated rx 155.89 ry -18.56 rz 54.57 deg; joints [-0.384, -42.528, 133.556, -159.618, 75.174, 60.735, 110.105]
  MoveL 805 to (-200.08, 75.42, -8.41) mm, rotated rx 156.06 ry -18.79 rz 54.04 deg; joints [-0.159, -42.966, 133.56, -159.124, 74.806, 60.697, 110.655]
  MoveL 806 to (-197.85, 75.42, -8.4) mm, rotated rx 156.13 ry -18.87 rz 53.83 deg; joints [-0.135, -43.13, 133.561, -158.996, 74.668, 60.682, 110.868]
  MoveL 807 to (-197.85, 75.42, -4.14) mm, rotated rx 156.13 ry -18.87 rz 53.83 deg; joints [0.086, -43.128, 133.553, -158.775, 74.662, 60.681, 110.868]
  Set speed (38.1 mm/s)
  MoveL 808 to (-197.89, 75.42, -3.98) mm, rotated rx 156.13 ry -18.87 rz 53.84 deg; joints [0.093, -43.125, 133.552, -158.769, 74.664, 60.681, 110.864]
  MoveL 809 to (-198.05, 75.11, -3.7) mm, rotated rx 156.1 ry -18.83 rz 53.93 deg; joints [0.097, -43.123, 133.571, -158.807, 74.677, 60.669, 110.768]
  Set speed (76.2 mm/s)
  MoveL 810 to (-198.05, 72.57, -3.7) mm, rotated rx 155.9 ry -18.57 rz 54.55 deg; joints [0.025, -43.2, 133.724, -159.155, 74.702, 60.561, 110.123]
  Set speed (38.1 mm/s)
  MoveL 811 to (-197.89, 72.25, -3.98) mm, rotated rx 155.88 ry -18.54 rz 54.61 deg; joints [0.004, -43.222, 133.744, -159.204, 74.695, 60.546, 110.057]
  MoveL 812 to (-197.85, 72.25, -4.14) mm, rotated rx 155.88 ry -18.55 rz 54.61 deg; joints [-0.004, -43.225, 133.745, -159.21, 74.693, 60.546, 110.061]
  Set speed (76.2 mm/s)
  MoveL 813 to (-197.85, 72.25, -8.4) mm, rotated rx 155.88 ry -18.55 rz 54.61 deg; joints [-0.225, -43.227, 133.752, -159.431, 74.699, 60.546, 110.061]
  MoveL 814 to (-200.08, 72.25, -8.41) mm, rotated rx 155.82 ry -18.46 rz 54.81 deg; joints [-0.249, -43.062, 133.75, -159.557, 74.836, 60.562, 109.854]
  MoveL 815 to (-206.05, 72.25, -11.57) mm, rotated rx 155.66 ry -18.24 rz 55.32 deg; joints [-0.473, -42.622, 133.742, -160.043, 75.203, 60.603, 109.323]
  MoveL 816 to (-201.08, 72.25, -20.25) mm, rotated rx 155.79 ry -18.42 rz 54.9 deg; joints [-0.872, -42.993, 133.763, -160.224, 74.91, 60.565, 109.764]
  MoveL 817 to (-201.08, 69.07, -20.25) mm, rotated rx 155.55 ry -18.09 rz 55.67 deg; joints [-0.966, -43.088, 133.953, -160.665, 74.938, 60.432, 108.959]
  MoveL 818 to (-206.05, 69.07, -11.57) mm, rotated rx 155.42 ry -17.92 rz 56.08 deg; joints [-0.564, -42.717, 133.929, -160.477, 75.231, 60.474, 108.533]
  MoveL 819 to (-200.08, 69.07, -8.41) mm, rotated rx 155.57 ry -18.13 rz 55.59 deg; joints [-0.341, -43.158, 133.941, -159.998, 74.865, 60.43, 109.046]
  MoveL 820 to (-197.85, 69.07, -8.4) mm, rotated rx 155.63 ry -18.21 rz 55.39 deg; joints [-0.317, -43.324, 133.945, -159.875, 74.729, 60.413, 109.246]
  MoveL 821 to (-197.85, 69.07, -4.14) mm, rotated rx 155.63 ry -18.21 rz 55.39 deg; joints [-0.096, -43.322, 133.938, -159.654, 74.723, 60.413, 109.246]
  Set speed (38.1 mm/s)
  MoveL 822 to (-197.89, 69.07, -3.98) mm, rotated rx 155.63 ry -18.21 rz 55.4 deg; joints [-0.088, -43.319, 133.938, -159.648, 74.725, 60.414, 109.242]
  MoveL 823 to (-198.05, 68.76, -3.7) mm, rotated rx 155.6 ry -18.17 rz 55.49 deg; joints [-0.085, -43.316, 133.956, -159.687, 74.737, 60.402, 109.146]
  Set speed (76.2 mm/s)
  MoveL 824 to (-198.05, 66.22, -3.7) mm, rotated rx 155.41 ry -17.9 rz 56.12 deg; joints [-0.161, -43.394, 134.112, -160.049, 74.76, 60.299, 108.487]
  Set speed (38.1 mm/s)
  MoveL 825 to (-197.89, 65.9, -3.98) mm, rotated rx 155.39 ry -17.87 rz 56.19 deg; joints [-0.183, -43.415, 134.132, -160.101, 74.753, 60.285, 108.418]
  MoveL 826 to (-197.85, 65.9, -4.14) mm, rotated rx 155.39 ry -17.87 rz 56.18 deg; joints [-0.191, -43.419, 134.133, -160.107, 74.751, 60.284, 108.422]
  Set speed (76.2 mm/s)
  MoveL 827 to (-197.85, 65.9, -8.4) mm, rotated rx 155.39 ry -17.87 rz 56.18 deg; joints [-0.412, -43.42, 134.139, -160.328, 74.757, 60.283, 108.422]
  MoveL 828 to (-200.08, 65.9, -8.41) mm, rotated rx 155.33 ry -17.79 rz 56.37 deg; joints [-0.435, -43.254, 134.134, -160.447, 74.893, 60.301, 108.23]
  MoveL 829 to (-206.05, 65.9, -11.57) mm, rotated rx 155.19 ry -17.58 rz 56.84 deg; joints [-0.658, -42.811, 134.117, -160.918, 75.257, 60.347, 107.736]
  MoveL 830 to (-201.08, 65.9, -20.25) mm, rotated rx 155.31 ry -17.75 rz 56.45 deg; joints [-1.061, -43.183, 134.143, -161.114, 74.965, 60.302, 108.146]
  MoveL 831 to (-201.08, 62.72, -20.25) mm, rotated rx 155.07 ry -17.41 rz 57.23 deg; joints [-1.159, -43.279, 134.334, -161.571, 74.989, 60.176, 107.325]
  MoveL 832 to (-206.05, 62.72, -11.57) mm, rotated rx 154.96 ry -17.24 rz 57.6 deg; joints [-0.754, -42.904, 134.306, -161.367, 75.281, 60.224, 106.931]
  MoveL 833 to (-200.08, 62.72, -8.41) mm, rotated rx 155.1 ry -17.44 rz 57.15 deg; joints [-0.532, -43.35, 134.327, -160.906, 74.919, 60.176, 107.406]
  MoveL 834 to (-197.85, 62.72, -8.4) mm, rotated rx 155.15 ry -17.52 rz 56.97 deg; joints [-0.51, -43.517, 134.335, -160.79, 74.783, 60.157, 107.591]
  MoveL 835 to (-197.85, 62.72, -4.14) mm, rotated rx 155.15 ry -17.52 rz 56.97 deg; joints [-0.288, -43.515, 134.328, -160.568, 74.777, 60.158, 107.591]
  Set speed (38.1 mm/s)
  MoveL 836 to (-197.89, 62.72, -3.98) mm, rotated rx 155.15 ry -17.52 rz 56.98 deg; joints [-0.28, -43.512, 134.328, -160.562, 74.78, 60.159, 107.587]
  MoveL 837 to (-198.05, 62.41, -3.7) mm, rotated rx 155.12 ry -17.48 rz 57.07 deg; joints [-0.277, -43.51, 134.347, -160.603, 74.792, 60.148, 107.49]
  Set speed (76.2 mm/s)
  MoveL 838 to (-198.05, 59.87, -3.7) mm, rotated rx 154.93 ry -17.2 rz 57.71 deg; joints [-0.356, -43.587, 134.504, -160.978, 74.811, 60.05, 106.82]
  Set speed (38.1 mm/s)
  MoveL 839 to (-197.89, 59.55, -3.98) mm, rotated rx 154.91 ry -17.17 rz 57.78 deg; joints [-0.379, -43.608, 134.525, -161.032, 74.804, 60.036, 106.748]
  MoveL 840 to (-197.85, 59.55, -4.14) mm, rotated rx 154.91 ry -17.17 rz 57.77 deg; joints [-0.387, -43.612, 134.525, -161.038, 74.802, 60.036, 106.751]
  Set speed (76.2 mm/s)
  MoveL 841 to (-197.85, 59.55, -8.4) mm, rotated rx 154.91 ry -17.17 rz 57.77 deg; joints [-0.61, -43.613, 134.531, -161.26, 74.807, 60.034, 106.751]
  MoveL 842 to (-200.08, 59.55, -8.41) mm, rotated rx 154.86 ry -17.09 rz 57.94 deg; joints [-0.631, -43.445, 134.522, -161.372, 74.943, 60.054, 106.574]
  MoveL 843 to (-206.05, 59.55, -11.57) mm, rotated rx 154.74 ry -16.9 rz 58.37 deg; joints [-0.852, -42.998, 134.495, -161.824, 75.304, 60.104, 106.12]
  MoveL 844 to (-201.08, 59.55, -20.25) mm, rotated rx 154.84 ry -17.06 rz 58.01 deg; joints [-1.26, -43.374, 134.527, -162.038, 75.012, 60.053, 106.497]
  MoveL 845 to (-201.08, 56.38, -20.25) mm, rotated rx 154.61 ry -16.7 rz 58.8 deg; joints [-1.362, -43.468, 134.72, -162.512, 75.033, 59.933, 105.662]
  MoveL 846 to (-206.05, 56.38, -11.57) mm, rotated rx 154.51 ry -16.55 rz 59.14 deg; joints [-0.952, -43.091, 134.686, -162.289, 75.325, 59.988, 105.302]
  MoveL 847 to (-200.08, 56.38, -8.41) mm, rotated rx 154.63 ry -16.73 rz 58.73 deg; joints [-0.733, -43.541, 134.717, -161.848, 74.965, 59.936, 105.736]
  MoveL 848 to (-197.85, 56.38, -8.4) mm, rotated rx 154.68 ry -16.81 rz 58.57 deg; joints [-0.712, -43.709, 134.728, -161.739, 74.83, 59.914, 105.905]
  MoveL 849 to (-197.85, 56.38, -4.14) mm, rotated rx 154.68 ry -16.81 rz 58.57 deg; joints [-0.489, -43.708, 134.723, -161.517, 74.825, 59.917, 105.905]
  Set speed (38.1 mm/s)
  MoveL 850 to (-197.89, 56.38, -3.98) mm, rotated rx 154.68 ry -16.8 rz 58.58 deg; joints [-0.481, -43.705, 134.723, -161.511, 74.827, 59.917, 105.901]
  MoveL 851 to (-198.05, 56.06, -3.7) mm, rotated rx 154.65 ry -16.76 rz 58.67 deg; joints [-0.478, -43.702, 134.741, -161.553, 74.839, 59.908, 105.804]
  Set speed (76.2 mm/s)
  MoveL 852 to (-198.05, 53.52, -3.7) mm, rotated rx 154.47 ry -16.47 rz 59.31 deg; joints [-0.562, -43.779, 134.9, -161.942, 74.855, 59.816, 105.122]
  Set speed (38.1 mm/s)
  MoveL 853 to (-197.89, 53.2, -3.98) mm, rotated rx 154.45 ry -16.44 rz 59.38 deg; joints [-0.585, -43.801, 134.921, -161.998, 74.848, 59.803, 105.048]
  MoveL 854 to (-197.85, 53.2, -4.14) mm, rotated rx 154.45 ry -16.44 rz 59.38 deg; joints [-0.593, -43.804, 134.921, -162.004, 74.845, 59.802, 105.051]
  Set speed (76.2 mm/s)
  MoveL 855 to (-197.85, 53.2, -8.4) mm, rotated rx 154.45 ry -16.44 rz 59.38 deg; joints [-0.817, -43.805, 134.926, -162.227, 74.85, 59.799, 105.051]
  MoveL 856 to (-200.08, 53.2, -8.41) mm, rotated rx 154.4 ry -16.37 rz 59.53 deg; joints [-0.837, -43.636, 134.913, -162.331, 74.985, 59.821, 104.89]
  MoveL 857 to (-206.05, 53.2, -11.57) mm, rotated rx 154.3 ry -16.19 rz 59.92 deg; joints [-1.055, -43.184, 134.877, -162.762, 75.344, 59.875, 104.477]
  MoveL 858 to (-201.08, 53.2, -20.25) mm, rotated rx 154.39 ry -16.34 rz 59.6 deg; joints [-1.468, -43.563, 134.913, -162.994, 75.052, 59.817, 104.82]
  MoveL 859 to (-201.08, 50.03, -20.25) mm, rotated rx 154.16 ry -15.97 rz 60.39 deg; joints [-1.575, -43.657, 135.108, -163.485, 75.069, 59.705, 103.971]
  MoveL 860 to (-206.05, 50.03, -11.57) mm, rotated rx 154.08 ry -15.83 rz 60.69 deg; joints [-1.16, -43.277, 135.068, -163.243, 75.362, 59.766, 103.647]
  MoveL 861 to (-200.08, 50.03, -8.41) mm, rotated rx 154.18 ry -16 rz 60.33 deg; joints [-0.944, -43.731, 135.11, -162.822, 75.003, 59.71, 104.038]
  MoveL 862 to (-197.85, 50.03, -8.4) mm, rotated rx 154.22 ry -16.07 rz 60.19 deg; joints [-0.924, -43.901, 135.125, -162.723, 74.868, 59.687, 104.19]
  MoveL 863 to (-197.85, 50.03, -4.14) mm, rotated rx 154.22 ry -16.07 rz 60.19 deg; joints [-0.7, -43.9, 135.121, -162.5, 74.864, 59.691, 104.19]
  Set speed (38.1 mm/s)
  MoveL 864 to (-197.89, 50.03, -3.98) mm, rotated rx 154.22 ry -16.07 rz 60.19 deg; joints [-0.692, -43.897, 135.12, -162.493, 74.866, 59.692, 104.187]
  MoveL 865 to (-197.93, 49.74, -3.64) mm, rotated rx 154.2 ry -16.03 rz 60.27 deg; joints [-0.684, -43.902, 135.138, -162.523, 74.87, 59.682, 104.106]
  Set speed (76.2 mm/s)
  MoveL 866 to (-196.9, 47.14, -3.04) mm, rotated rx 154.03 ry -15.75 rz 60.87 deg; joints [-0.733, -44.06, 135.307, -162.858, 74.821, 59.584, 103.464]
  Set speed (38.1 mm/s)
  MoveL 867 to (-196.62, 46.85, -3.25) mm, rotated rx 154.02 ry -15.72 rz 60.92 deg; joints [-0.752, -44.09, 135.328, -162.904, 74.806, 59.572, 103.402]
  MoveL 868 to (-195.49, 46.85, -5.2) mm, rotated rx 154.04 ry -15.76 rz 60.85 deg; joints [-0.845, -44.176, 135.337, -162.957, 74.74, 59.557, 103.477]
  MoveL 869 to (-195.45, 46.85, -5.36) mm, rotated rx 154.04 ry -15.76 rz 60.85 deg; joints [-0.853, -44.18, 135.337, -162.963, 74.737, 59.557, 103.48]
  Set speed (76.2 mm/s)
  MoveL 870 to (-195.45, 46.85, -9.71) mm, rotated rx 154.04 ry -15.76 rz 60.85 deg; joints [-1.082, -44.181, 135.34, -163.191, 74.741, 59.553, 103.48]
  MoveL 871 to (-203.6, 46.85, -10.15) mm, rotated rx 153.91 ry -15.53 rz 61.34 deg; joints [-1.173, -43.557, 135.28, -163.558, 75.23, 59.638, 102.959]
  MoveL 872 to (-198.68, 46.85, -18.86) mm, rotated rx 153.99 ry -15.66 rz 61.05 deg; joints [-1.592, -43.935, 135.321, -163.81, 74.939, 59.576, 103.269]
  Set speed (38.1 mm/s)
  MoveL 873 to (-199.55, 46.85, -18.63) mm, rotated rx 153.97 ry -15.64 rz 61.1 deg; joints [-1.587, -43.869, 135.314, -163.834, 74.992, 59.584, 103.213]
  Set speed (100.0 mm/s)
  MoveL 874 to (-233.61, 46.85, 40.17) mm, rotated rx 153.51 ry -14.81 rz 62.84 deg; joints [1.28, -41.218, 134.842, -162.004, 76.852, 60.082, 101.34]
  Print: /'Cut out part'
  Set speed (100.0 mm/s)
  MoveL 875 to (-197.68, 45.77, 34.52) mm, rotated rx -180 ry 0 rz 65.64 deg; joints [-1.565, -54.082, 140.719, -180.026, 73.937, 89.925, 103.036]
  MoveL 876 to (-197.68, 45.77, 3.11) mm, rotated rx 180 ry 0 rz 65.64 deg; joints [-3.293, -54.076, 140.683, -181.781, 73.909, 90.031, 103.036]
  Set speed (25.4 mm/s)
  MoveL 877 to (-197.68, 45.77, -0.84) mm, rotated rx -180 ry 0 rz 65.64 deg; joints [-3.51, -54.073, 140.674, -182.001, 73.902, 90.045, 103.036]
  MoveL 878 to (-197.57, 46.4, -1.48) mm, rotated rx 180 ry 0 rz 65.46 deg; joints [-3.545, -54.07, 140.672, -182.036, 73.904, 90.047, 103.215]
  Set speed (38.1 mm/s)
  MoveL 879 to (-197.51, 46.74, -1.47) mm, rotated rx 180 ry 0 rz 65.37 deg; joints [-3.545, -54.068, 140.671, -182.036, 73.905, 90.047, 103.314]
  MoveL 880 to (-196.6, 47.2, -1.48) mm, rotated rx 180 ry 0 rz 65.18 deg; joints [-3.545, -54.135, 140.68, -182.037, 73.847, 90.049, 103.501]
  Set speed (76.2 mm/s)
  MoveL 881 to (-196.42, 47.11, -1.48) mm, rotated rx 180 ry 0 rz 65.19 deg; joints [-3.545, -54.152, 140.682, -182.037, 73.832, 90.05, 103.488]
  MoveL 882 to (-196.18, 47.01, -1.47) mm, rotated rx -180 ry 0 rz 65.2 deg; joints [-3.544, -54.174, 140.685, -182.037, 73.813, 90.05, 103.477]
  MoveL 883 to (-195.93, 46.94, -1.48) mm, rotated rx -180 ry 0 rz 65.21 deg; joints [-3.544, -54.195, 140.688, -182.037, 73.794, 90.051, 103.472]
  MoveL 884 to (-195.69, 46.88, -1.48) mm, rotated rx -180 ry 0 rz 65.21 deg; joints [-3.544, -54.217, 140.691, -182.038, 73.776, 90.052, 103.472]
  MoveL 885 to (-195.45, 46.84, -1.47) mm, rotated rx -180 ry 0 rz 65.2 deg; joints [-3.544, -54.238, 140.693, -182.038, 73.758, 90.052, 103.478]
  MoveL 886 to (-195.21, 46.83, -1.47) mm, rotated rx 180 ry 0 rz 65.19 deg; joints [-3.544, -54.258, 140.696, -182.038, 73.74, 90.053, 103.489]
  MoveL 887 to (-194.97, 46.83, -1.48) mm, rotated rx -180 ry 0 rz 65.18 deg; joints [-3.544, -54.278, 140.698, -182.038, 73.722, 90.054, 103.505]
  MoveL 888 to (213.41, 46.82, -1.47) mm, rotated rx -180 ry 0 rz -48.94 deg; joints [-3.719, -87.202, 145.334, -190.983, 6.914, 99.143, 179]
  MoveL 889 to (213.89, 46.83, -1.47) mm, rotated rx 180 ry 0 rz -48.97 deg; joints [-3.72, -87.233, 145.356, -191.035, 6.88, 99.194, 179]
  MoveL 890 to (214.13, 46.85, -1.47) mm, rotated rx 180 ry 0 rz -48.98 deg; joints [-3.72, -87.247, 145.37, -191.048, 6.873, 99.207, 179]
  MoveL 891 to (214.37, 46.9, -1.48) mm, rotated rx 180 ry 0 rz -48.98 deg; joints [-3.721, -87.26, 145.386, -191.049, 6.873, 99.207, 179]
  MoveL 892 to (214.63, 46.96, -1.48) mm, rotated rx -180 ry 0 rz -48.98 deg; joints [-3.721, -87.273, 145.407, -191.037, 6.883, 99.195, 179]
  MoveL 893 to (214.88, 47.05, -1.48) mm, rotated rx 180 ry 0 rz -48.97 deg; joints [-3.722, -87.284, 145.43, -191.01, 6.904, 99.167, 179]
  MoveL 894 to (215.01, 47.11, -1.48) mm, rotated rx -180 ry 0 rz -48.96 deg; joints [-3.722, -87.289, 145.443, -190.991, 6.918, 99.147, 179]
  MoveL 895 to (215.14, 47.17, -1.48) mm, rotated rx -180 ry 0 rz -48.95 deg; joints [-3.723, -87.294, 145.457, -190.967, 6.935, 99.124, 179]
  MoveL 896 to (215.26, 47.23, -1.48) mm, rotated rx -180 ry 0 rz -48.94 deg; joints [-3.723, -87.298, 145.471, -190.94, 6.956, 99.096, 179]
  MoveL 897 to (215.39, 47.31, -1.47) mm, rotated rx 180 ry 0 rz -48.93 deg; joints [-3.724, -87.301, 145.487, -190.907, 6.98, 99.063, 179]
  MoveL 898 to (215.62, 47.47, -1.48) mm, rotated rx 180 ry 0 rz -48.91 deg; joints [-3.724, -87.307, 145.518, -190.838, 7.032, 98.992, 179]
  MoveL 899 to (215.84, 47.66, -1.48) mm, rotated rx -180 ry 0 rz -48.87 deg; joints [-3.725, -87.31, 145.553, -190.75, 7.098, 98.904, 179]
  MoveL 900 to (215.98, 47.78, -1.48) mm, rotated rx -180 ry 0 rz -48.84 deg; joints [-3.726, -87.31, 145.576, -190.688, 7.144, 98.842, 179]
  MoveL 901 to (216.1, 47.91, -1.47) mm, rotated rx 180 ry 0 rz -48.82 deg; joints [-3.727, -87.31, 145.598, -190.626, 7.192, 98.779, 179]
  MoveL 902 to (216.2, 48.04, -1.47) mm, rotated rx -180 ry 0 rz -48.79 deg; joints [-3.727, -87.309, 145.62, -190.564, 7.241, 98.716, 179]
  MoveL 903 to (216.3, 48.17, -1.48) mm, rotated rx 180 ry 0 rz -48.77 deg; joints [-3.728, -87.307, 145.641, -190.501, 7.291, 98.653, 179]
  MoveL 904 to (216.39, 48.31, -1.48) mm, rotated rx -180 ry 0 rz -48.74 deg; joints [-3.728, -87.305, 145.663, -190.436, 7.343, 98.587, 179]
  MoveL 905 to (216.47, 48.44, -1.48) mm, rotated rx -180 ry 0 rz -48.71 deg; joints [-3.729, -87.302, 145.684, -190.37, 7.396, 98.522, 179]
  MoveL 906 to (216.54, 48.57, -1.47) mm, rotated rx 180 ry 0 rz -48.68 deg; joints [-3.729, -87.298, 145.704, -190.305, 7.449, 98.456, 179]
  MoveL 907 to (216.6, 48.71, -1.47) mm, rotated rx 180 ry 0 rz -48.65 deg; joints [-3.73, -87.294, 145.725, -190.24, 7.503, 98.39, 179]
  MoveL 908 to (216.66, 48.84, -1.47) mm, rotated rx -180 ry 0 rz -48.62 deg; joints [-3.73, -87.289, 145.745, -190.175, 7.558, 98.325, 179]
  MoveL 909 to (216.71, 48.97, -1.48) mm, rotated rx -180 ry 0 rz -48.59 deg; joints [-3.731, -87.283, 145.764, -190.111, 7.613, 98.26, 179]
  MoveL 910 to (216.75, 49.11, -1.48) mm, rotated rx 180 ry 0 rz -48.55 deg; joints [-3.731, -87.278, 145.784, -190.046, 7.669, 98.196, 179]
  MoveL 911 to (216.79, 49.24, -1.47) mm, rotated rx -180 ry 0 rz -48.52 deg; joints [-3.732, -87.271, 145.803, -189.982, 7.725, 98.131, 179]
  MoveL 912 to (216.84, 49.48, -1.47) mm, rotated rx 180 ry 0 rz -48.47 deg; joints [-3.732, -87.259, 145.837, -189.868, 7.828, 98.016, 179]
  MoveL 913 to (216.87, 49.73, -1.48) mm, rotated rx -180 ry 0 rz -48.41 deg; joints [-3.733, -87.246, 145.869, -189.755, 7.932, 97.903, 179]
  MoveL 914 to (216.88, 49.97, -1.47) mm, rotated rx 180 ry 0 rz -48.35 deg; joints [-3.734, -87.231, 145.901, -189.643, 8.037, 97.79, 179]
  MoveL 915 to (216.87, 50.21, -1.48) mm, rotated rx 180 ry 0 rz -48.29 deg; joints [-3.735, -87.214, 145.932, -189.532, 8.144, 97.679, 179]
  MoveL 916 to (216.85, 50.45, -1.47) mm, rotated rx -180 ry 0 rz -48.22 deg; joints [-3.735, -87.197, 145.962, -189.423, 8.253, 97.569, 179]
  MoveL 917 to (216.8, 50.69, -1.48) mm, rotated rx -180 ry 0 rz -48.16 deg; joints [-3.736, -87.178, 145.992, -189.315, 8.363, 97.46, 179]
  MoveL 918 to (216.74, 50.93, -1.48) mm, rotated rx -180 ry 0 rz -48.1 deg; joints [-3.736, -87.158, 146.02, -189.208, 8.475, 97.353, 179]
  MoveL 919 to (216.65, 51.18, -1.47) mm, rotated rx -180 ry 0 rz -48.03 deg; joints [-3.737, -87.136, 146.048, -189.102, 8.589, 97.247, 179]
  MoveL 920 to (216.58, 51.34, -1.47) mm, rotated rx -180 ry 0 rz -47.99 deg; joints [-3.737, -87.12, 146.065, -189.031, 8.667, 97.175, 179]
  MoveL 921 to (216.5, 51.5, -1.48) mm, rotated rx -180 ry 0 rz -47.94 deg; joints [-3.738, -87.104, 146.083, -188.96, 8.746, 97.104, 179]
  MoveL 922 to (216.41, 51.67, -1.47) mm, rotated rx -180 ry 0 rz -47.89 deg; joints [-3.738, -87.087, 146.1, -188.889, 8.826, 97.033, 179]
  MoveL 923 to (216.3, 51.83, -1.48) mm, rotated rx -180 ry 0 rz -47.85 deg; joints [-3.738, -87.068, 146.116, -188.819, 8.907, 96.963, 179]
  MoveL 924 to (216.2, 51.96, -1.47) mm, rotated rx 180 ry 0 rz -47.81 deg; joints [-3.738, -87.053, 146.129, -188.761, 8.975, 96.904, 179]
  MoveL 925 to (216.09, 52.1, -1.48) mm, rotated rx -180 ry 0 rz -47.76 deg; joints [-3.739, -87.036, 146.142, -188.702, 9.044, 96.846, 179]
  MoveL 926 to (215.96, 52.23, -1.48) mm, rotated rx -180 ry 0 rz -47.72 deg; joints [-3.739, -87.018, 146.154, -188.644, 9.115, 96.788, 179]
  MoveL 927 to (215.82, 52.37, -1.47) mm, rotated rx 180 ry 0 rz -47.68 deg; joints [-3.739, -87, 146.165, -188.585, 9.186, 96.729, 179]
  MoveL 928 to (215.58, 52.56, -1.47) mm, rotated rx -180 ry 0 rz -47.62 deg; joints [-3.739, -86.97, 146.179, -188.5, 9.293, 96.643, 179]
  MoveL 929 to (215.34, 52.72, -1.48) mm, rotated rx -180 ry 0 rz -47.56 deg; joints [-3.739, -86.943, 146.19, -188.428, 9.384, 96.571, 179]
  MoveL 930 to (215.09, 52.85, -1.47) mm, rotated rx 180 ry 0 rz -47.51 deg; joints [-3.739, -86.918, 146.196, -188.367, 9.463, 96.51, 179]
  MoveL 931 to (214.85, 52.96, -1.48) mm, rotated rx -180 ry 0 rz -47.47 deg; joints [-3.739, -86.895, 146.199, -188.315, 9.53, 96.459, 179]
  MoveL 932 to (214.61, 53.04, -1.48) mm, rotated rx -180 ry 0 rz -47.44 deg; joints [-3.739, -86.873, 146.199, -188.272, 9.587, 96.415, 179]
  MoveL 933 to (214.37, 53.1, -1.48) mm, rotated rx 180 ry 0 rz -47.41 deg; joints [-3.739, -86.853, 146.197, -188.235, 9.635, 96.379, 179]
  MoveL 934 to (214.36, 53.11, -1.47) mm, rotated rx -180 ry 0 rz -47.41 deg; joints [-3.739, -86.851, 146.197, -188.233, 9.638, 96.377, 179]
  MoveL 935 to (214.12, 53.15, -1.48) mm, rotated rx -180 ry 0 rz -47.38 deg; joints [-3.738, -86.833, 146.192, -188.204, 9.677, 96.348, 179]
  MoveL 936 to (213.88, 53.17, -1.48) mm, rotated rx -180 ry 0 rz -47.36 deg; joints [-3.738, -86.815, 146.184, -188.181, 9.707, 96.325, 179]
  MoveL 937 to (213.4, 53.17, -1.48) mm, rotated rx -180 ry 0 rz -47.33 deg; joints [-3.737, -86.783, 146.164, -188.147, 9.75, 96.293, 179]
  MoveL 938 to (-195.12, 53.17, -1.48) mm, rotated rx -180 ry 0 rz 63.44 deg; joints [-3.545, -54.131, 140.68, -182.037, 73.851, 90.049, 105.244]
  MoveL 939 to (-195.28, 53.17, -1.48) mm, rotated rx -180 ry 0 rz 63.45 deg; joints [-3.545, -54.118, 140.678, -182.037, 73.862, 90.049, 105.231]
  MoveL 940 to (-195.43, 53.16, -1.48) mm, rotated rx 180 ry 0 rz 63.46 deg; joints [-3.545, -54.105, 140.676, -182.037, 73.873, 90.048, 105.216]
  MoveL 941 to (-195.59, 53.14, -1.48) mm, rotated rx -180 ry 0 rz 63.48 deg; joints [-3.545, -54.092, 140.675, -182.037, 73.884, 90.048, 105.199]
  MoveL 942 to (-195.75, 53.11, -1.48) mm, rotated rx -180 ry 0 rz 63.5 deg; joints [-3.545, -54.08, 140.673, -182.037, 73.895, 90.047, 105.179]
  MoveL 943 to (-195.92, 53.07, -1.47) mm, rotated rx 180 ry 0 rz 63.52 deg; joints [-3.545, -54.067, 140.671, -182.036, 73.906, 90.047, 105.156]
  MoveL 944 to (-196.08, 53.02, -1.47) mm, rotated rx 180 ry 0 rz 63.55 deg; joints [-3.545, -54.054, 140.67, -182.036, 73.917, 90.047, 105.13]
  MoveL 945 to (-196.25, 52.96, -1.47) mm, rotated rx 180 ry 0 rz 63.58 deg; joints [-3.545, -54.042, 140.668, -182.036, 73.928, 90.046, 105.102]
  MoveL 946 to (-196.42, 52.89, -1.47) mm, rotated rx -180 ry 0 rz 63.61 deg; joints [-3.545, -54.029, 140.666, -182.036, 73.939, 90.046, 105.07]
  MoveL 947 to (-196.56, 52.82, -1.48) mm, rotated rx 180 ry 0 rz 63.64 deg; joints [-3.545, -54.019, 140.665, -182.036, 73.948, 90.045, 105.041]
  MoveL 948 to (-196.7, 52.74, -1.47) mm, rotated rx 180 ry 0 rz 63.67 deg; joints [-3.545, -54.009, 140.664, -182.036, 73.956, 90.045, 105.01]
  MoveL 949 to (-196.84, 52.66, -1.47) mm, rotated rx 180 ry 0 rz 63.7 deg; joints [-3.545, -54, 140.662, -182.036, 73.965, 90.045, 104.977]
  MoveL 950 to (-196.98, 52.56, -1.47) mm, rotated rx 180 ry 0 rz 63.74 deg; joints [-3.545, -53.99, 140.661, -182.036, 73.973, 90.044, 104.94]
  MoveL 951 to (-197.12, 52.45, -1.47) mm, rotated rx 180 ry 0 rz 63.78 deg; joints [-3.545, -53.981, 140.66, -182.036, 73.981, 90.044, 104.9]
  MoveL 952 to (-197.26, 52.33, -1.48) mm, rotated rx 180 ry 0 rz 63.82 deg; joints [-3.545, -53.972, 140.659, -182.036, 73.988, 90.044, 104.857]
  MoveL 953 to (-197.41, 52.18, -1.48) mm, rotated rx -180 ry 0 rz 63.87 deg; joints [-3.545, -53.963, 140.658, -182.036, 73.996, 90.044, 104.806]
  MoveL 954 to (-197.54, 52.03, -1.48) mm, rotated rx 180 ry 0 rz 63.92 deg; joints [-3.545, -53.955, 140.657, -182.036, 74.003, 90.043, 104.757]
  MoveL 955 to (-197.7, 51.82, -1.48) mm, rotated rx 180 ry 0 rz 63.99 deg; joints [-3.545, -53.946, 140.655, -182.036, 74.011, 90.043, 104.687]
  MoveL 956 to (-197.84, 51.6, -1.48) mm, rotated rx -180 ry 0 rz 64.06 deg; joints [-3.545, -53.94, 140.655, -182.035, 74.017, 90.043, 104.619]
  MoveL 957 to (-197.95, 51.39, -1.47) mm, rotated rx 180 ry 0 rz 64.13 deg; joints [-3.545, -53.935, 140.654, -182.035, 74.021, 90.043, 104.553]
  MoveL 958 to (-198.05, 51.18, -1.47) mm, rotated rx 180 ry 0 rz 64.19 deg; joints [-3.545, -53.931, 140.653, -182.035, 74.024, 90.043, 104.488]
  MoveL 959 to (-198.13, 50.93, -1.48) mm, rotated rx 180 ry 0 rz 64.26 deg; joints [-3.545, -53.93, 140.653, -182.035, 74.025, 90.043, 104.417]
  MoveL 960 to (-198.2, 50.69, -1.47) mm, rotated rx 180 ry 0 rz 64.33 deg; joints [-3.545, -53.929, 140.653, -182.035, 74.025, 90.043, 104.347]
  MoveL 961 to (-198.24, 50.45, -1.47) mm, rotated rx 180 ry 0 rz 64.4 deg; joints [-3.545, -53.931, 140.653, -182.035, 74.024, 90.043, 104.278]
  MoveL 962 to (-198.27, 50.21, -1.48) mm, rotated rx 180 ry 0 rz 64.47 deg; joints [-3.545, -53.934, 140.654, -182.035, 74.022, 90.043, 104.211]
  MoveL 963 to (-198.27, 49.97, -1.48) mm, rotated rx -180 ry 0 rz 64.53 deg; joints [-3.545, -53.938, 140.654, -182.035, 74.018, 90.043, 104.145]
  MoveL 964 to (-198.26, 49.73, -1.48) mm, rotated rx -180 ry 0 rz 64.6 deg; joints [-3.545, -53.944, 140.655, -182.035, 74.012, 90.043, 104.08]
  MoveL 965 to (-198.23, 49.48, -1.48) mm, rotated rx 180 ry 0 rz 64.66 deg; joints [-3.545, -53.952, 140.656, -182.036, 74.006, 90.043, 104.016]
  MoveL 966 to (-198.18, 49.24, -1.47) mm, rotated rx -180 ry 0 rz 64.73 deg; joints [-3.545, -53.961, 140.657, -182.036, 73.998, 90.044, 103.954]
  MoveL 967 to (-198.11, 49, -1.48) mm, rotated rx 180 ry 0 rz 64.79 deg; joints [-3.545, -53.972, 140.659, -182.036, 73.989, 90.044, 103.893]
  MoveL 968 to (-198.02, 48.76, -1.47) mm, rotated rx 180 ry 0 rz 64.85 deg; joints [-3.545, -53.984, 140.66, -182.036, 73.978, 90.044, 103.833]
  MoveL 969 to (-197.91, 48.52, -1.48) mm, rotated rx -180 ry 0 rz 64.9 deg; joints [-3.545, -53.999, 140.662, -182.036, 73.965, 90.045, 103.775]
  MoveL 970 to (-197.76, 48.28, -1.48) mm, rotated rx -180 ry 0 rz 64.96 deg; joints [-3.545, -54.016, 140.665, -182.036, 73.951, 90.045, 103.718]
  MoveL 971 to (-197.66, 48.13, -1.48) mm, rotated rx -180 ry 0 rz 64.99 deg; joints [-3.545, -54.027, 140.666, -182.036, 73.941, 90.046, 103.685]
  MoveL 972 to (-197.55, 47.98, -1.47) mm, rotated rx 180 ry 0 rz 65.03 deg; joints [-3.545, -54.04, 140.668, -182.036, 73.93, 90.046, 103.652]
  MoveL 973 to (-197.42, 47.84, -1.48) mm, rotated rx -180 ry 0 rz 65.06 deg; joints [-3.545, -54.053, 140.669, -182.036, 73.918, 90.046, 103.62]
  MoveL 974 to (-197.27, 47.69, -1.48) mm, rotated rx 180 ry 0 rz 65.09 deg; joints [-3.545, -54.069, 140.671, -182.036, 73.905, 90.047, 103.59]
  MoveL 975 to (-197.03, 47.48, -1.47) mm, rotated rx 180 ry 0 rz 65.13 deg; joints [-3.545, -54.093, 140.675, -182.037, 73.883, 90.048, 103.549]
  MoveL 976 to (-196.78, 47.31, -1.48) mm, rotated rx -180 ry 0 rz 65.16 deg; joints [-3.545, -54.117, 140.678, -182.037, 73.863, 90.049, 103.518]
  MoveL 977 to (-196.6, 47.2, -1.48) mm, rotated rx 180 ry 0 rz 65.18 deg; joints [-3.545, -54.135, 140.68, -182.037, 73.847, 90.049, 103.501]
  Set speed (38.1 mm/s)
  MoveL 978 to (-197.17, 46.07, -1.48) mm, rotated rx -180 ry 0 rz 65.53 deg; joints [-3.545, -54.11, 140.677, -182.037, 73.869, 90.048, 103.151]
  MoveL 979 to (-197.73, 46.35, -1.48) mm, rotated rx 180 ry 0 rz 65.49 deg; joints [-3.545, -54.057, 140.67, -182.036, 73.915, 90.047, 103.192]
  Set speed (25.4 mm/s)
  MoveL 980 to (-197.73, 46.35, -3.84) mm, rotated rx 180 ry 0 rz 65.49 deg; joints [-3.675, -54.055, 140.664, -182.168, 73.91, 90.055, 103.192]
  MoveL 981 to (-197.45, 46.92, -4.48) mm, rotated rx 180 ry 0 rz 65.31 deg; joints [-3.709, -54.067, 140.663, -182.204, 73.898, 90.057, 103.366]
  Set speed (38.1 mm/s)
  MoveL 982 to (-196.6, 47.2, -4.48) mm, rotated rx -180 ry 0 rz 65.18 deg; joints [-3.709, -54.133, 140.672, -182.204, 73.842, 90.06, 103.501]
  Set speed (76.2 mm/s)
  MoveL 983 to (-196.42, 47.11, -4.48) mm, rotated rx -180 ry 0 rz 65.19 deg; joints [-3.709, -54.15, 140.674, -182.205, 73.827, 90.06, 103.488]
  MoveL 984 to (-196.18, 47.01, -4.47) mm, rotated rx -180 ry 0 rz 65.2 deg; joints [-3.709, -54.172, 140.677, -182.205, 73.807, 90.061, 103.477]
  MoveL 985 to (-195.93, 46.94, -4.47) mm, rotated rx 180 ry 0 rz 65.21 deg; joints [-3.709, -54.194, 140.68, -182.205, 73.789, 90.062, 103.472]
  MoveL 986 to (-195.69, 46.88, -4.47) mm, rotated rx -180 ry 0 rz 65.21 deg; joints [-3.709, -54.215, 140.683, -182.205, 73.77, 90.063, 103.472]
  MoveL 987 to (-195.45, 46.84, -4.47) mm, rotated rx 180 ry 0 rz 65.2 deg; joints [-3.709, -54.236, 140.685, -182.205, 73.752, 90.063, 103.478]
  MoveL 988 to (-195.21, 46.83, -4.47) mm, rotated rx 180 ry 0 rz 65.19 deg; joints [-3.709, -54.256, 140.688, -182.205, 73.734, 90.064, 103.489]
  MoveL 989 to (-194.97, 46.82, -4.48) mm, rotated rx -180 ry 0 rz 65.18 deg; joints [-3.709, -54.276, 140.69, -182.206, 73.716, 90.065, 103.505]
  MoveL 990 to (213.41, 46.82, -4.47) mm, rotated rx -180 ry 0 rz -48.94 deg; joints [-3.9, -87.194, 145.325, -191.911, 6.932, 99.922, 179]
  MoveL 991 to (213.89, 46.83, -4.48) mm, rotated rx -180 ry 0 rz -48.97 deg; joints [-3.901, -87.225, 145.348, -191.967, 6.898, 99.978, 179]
  MoveL 992 to (214.13, 46.85, -4.48) mm, rotated rx -180 ry 0 rz -48.98 deg; joints [-3.901, -87.24, 145.362, -191.981, 6.891, 99.992, 179]
  MoveL 993 to (214.37, 46.9, -4.48) mm, rotated rx -180 ry 0 rz -48.98 deg; joints [-3.902, -87.253, 145.378, -191.982, 6.891, 99.992, 179]
  MoveL 994 to (214.63, 46.96, -4.48) mm, rotated rx -180 ry 0 rz -48.98 deg; joints [-3.903, -87.265, 145.398, -191.969, 6.901, 99.978, 179]
  MoveL 995 to (214.88, 47.05, -4.48) mm, rotated rx -180 ry 0 rz -48.97 deg; joints [-3.904, -87.277, 145.422, -191.94, 6.922, 99.949, 179]
  MoveL 996 to (215.01, 47.11, -4.47) mm, rotated rx -180 ry 0 rz -48.96 deg; joints [-3.904, -87.282, 145.434, -191.919, 6.936, 99.927, 179]
  MoveL 997 to (215.14, 47.17, -4.47) mm, rotated rx -180 ry 0 rz -48.95 deg; joints [-3.904, -87.286, 145.448, -191.894, 6.953, 99.902, 179]
  MoveL 998 to (215.26, 47.23, -4.47) mm, rotated rx -180 ry 0 rz -48.94 deg; joints [-3.905, -87.29, 145.463, -191.864, 6.974, 99.871, 179]
  MoveL 999 to (215.39, 47.31, -4.48) mm, rotated rx -180 ry 0 rz -48.93 deg; joints [-3.905, -87.294, 145.479, -191.829, 6.998, 99.836, 179]
  MoveL 1000 to (215.62, 47.47, -4.48) mm, rotated rx -180 ry 0 rz -48.91 deg; joints [-3.906, -87.299, 145.51, -191.754, 7.049, 99.76, 179]
  MoveL 1001 to (215.84, 47.66, -4.48) mm, rotated rx 180 ry 0 rz -48.87 deg; joints [-3.907, -87.302, 145.545, -191.658, 7.115, 99.664, 179]
  MoveL 1002 to (215.98, 47.78, -4.48) mm, rotated rx 180 ry 0 rz -48.84 deg; joints [-3.908, -87.303, 145.568, -191.592, 7.162, 99.597, 179]
  MoveL 1003 to (216.1, 47.91, -4.48) mm, rotated rx -180 ry 0 rz -48.82 deg; joints [-3.908, -87.303, 145.59, -191.525, 7.21, 99.529, 179]
  MoveL 1004 to (216.2, 48.04, -4.47) mm, rotated rx 180 ry 0 rz -48.79 deg; joints [-3.909, -87.302, 145.612, -191.457, 7.258, 99.461, 179]
  MoveL 1005 to (216.3, 48.17, -4.48) mm, rotated rx 180 ry 0 rz -48.77 deg; joints [-3.91, -87.3, 145.633, -191.389, 7.308, 99.393, 179]
  MoveL 1006 to (216.39, 48.31, -4.48) mm, rotated rx -180 ry 0 rz -48.74 deg; joints [-3.91, -87.297, 145.654, -191.319, 7.36, 99.322, 179]
  MoveL 1007 to (216.47, 48.44, -4.48) mm, rotated rx -180 ry 0 rz -48.71 deg; joints [-3.911, -87.294, 145.675, -191.248, 7.413, 99.25, 179]
  MoveL 1008 to (216.54, 48.57, -4.48) mm, rotated rx -180 ry 0 rz -48.68 deg; joints [-3.911, -87.29, 145.696, -191.178, 7.466, 99.179, 179]
  MoveL 1009 to (216.6, 48.71, -4.48) mm, rotated rx -180 ry 0 rz -48.65 deg; joints [-3.912, -87.286, 145.716, -191.107, 7.52, 99.109, 179]
  MoveL 1010 to (216.66, 48.84, -4.48) mm, rotated rx 180 ry 0 rz -48.62 deg; joints [-3.912, -87.281, 145.736, -191.037, 7.574, 99.038, 179]
  MoveL 1011 to (216.71, 48.97, -4.48) mm, rotated rx -180 ry 0 rz -48.59 deg; joints [-3.913, -87.276, 145.756, -190.967, 7.63, 98.968, 179]
  MoveL 1012 to (216.75, 49.11, -4.48) mm, rotated rx 180 ry 0 rz -48.55 deg; joints [-3.913, -87.27, 145.775, -190.898, 7.685, 98.898, 179]
  MoveL 1013 to (216.79, 49.24, -4.48) mm, rotated rx -180 ry 0 rz -48.52 deg; joints [-3.914, -87.264, 145.794, -190.828, 7.741, 98.828, 179]
  MoveL 1014 to (216.84, 49.48, -4.47) mm, rotated rx 180 ry 0 rz -48.47 deg; joints [-3.915, -87.252, 145.828, -190.705, 7.844, 98.704, 179]
  MoveL 1015 to (216.87, 49.73, -4.48) mm, rotated rx -180 ry 0 rz -48.41 deg; joints [-3.916, -87.238, 145.861, -190.582, 7.947, 98.581, 179]
  MoveL 1016 to (216.88, 49.97, -4.48) mm, rotated rx -180 ry 0 rz -48.35 deg; joints [-3.916, -87.223, 145.893, -190.461, 8.053, 98.459, 179]
  MoveL 1017 to (216.87, 50.21, -4.48) mm, rotated rx -180 ry 0 rz -48.29 deg; joints [-3.917, -87.207, 145.924, -190.341, 8.16, 98.338, 179]
  MoveL 1018 to (216.85, 50.45, -4.47) mm, rotated rx 180 ry 0 rz -48.22 deg; joints [-3.918, -87.189, 145.954, -190.223, 8.268, 98.219, 179]
  MoveL 1019 to (216.8, 50.69, -4.47) mm, rotated rx -180 ry 0 rz -48.16 deg; joints [-3.918, -87.171, 145.983, -190.106, 8.378, 98.102, 179]
  MoveL 1020 to (216.74, 50.93, -4.47) mm, rotated rx -180 ry 0 rz -48.1 deg; joints [-3.919, -87.15, 146.012, -189.99, 8.49, 97.985, 179]
  MoveL 1021 to (216.65, 51.17, -4.48) mm, rotated rx 180 ry 0 rz -48.03 deg; joints [-3.92, -87.129, 146.039, -189.875, 8.603, 97.87, 179]
  MoveL 1022 to (216.58, 51.34, -4.47) mm, rotated rx 180 ry 0 rz -47.99 deg; joints [-3.92, -87.113, 146.057, -189.798, 8.681, 97.793, 179]
  MoveL 1023 to (216.5, 51.5, -4.47) mm, rotated rx 180 ry 0 rz -47.94 deg; joints [-3.92, -87.097, 146.075, -189.721, 8.76, 97.716, 179]
  MoveL 1024 to (216.41, 51.67, -4.47) mm, rotated rx -180 ry 0 rz -47.89 deg; joints [-3.921, -87.079, 146.092, -189.645, 8.84, 97.639, 179]
  MoveL 1025 to (216.3, 51.83, -4.48) mm, rotated rx 180 ry 0 rz -47.85 deg; joints [-3.921, -87.061, 146.108, -189.568, 8.921, 97.563, 179]
  MoveL 1026 to (216.2, 51.96, -4.48) mm, rotated rx -180 ry 0 rz -47.81 deg; joints [-3.921, -87.045, 146.121, -189.505, 8.989, 97.499, 179]
  MoveL 1027 to (216.09, 52.1, -4.48) mm, rotated rx -180 ry 0 rz -47.76 deg; joints [-3.921, -87.028, 146.133, -189.442, 9.058, 97.436, 179]
  MoveL 1028 to (215.96, 52.23, -4.48) mm, rotated rx -180 ry 0 rz -47.72 deg; joints [-3.922, -87.011, 146.145, -189.379, 9.128, 97.373, 179]
  MoveL 1029 to (215.82, 52.37, -4.48) mm, rotated rx -180 ry 0 rz -47.68 deg; joints [-3.922, -86.992, 146.156, -189.315, 9.2, 97.309, 179]
  MoveL 1030 to (215.58, 52.56, -4.48) mm, rotated rx -180 ry 0 rz -47.62 deg; joints [-3.922, -86.963, 146.171, -189.222, 9.306, 97.216, 179]
  MoveL 1031 to (215.34, 52.72, -4.48) mm, rotated rx -180 ry 0 rz -47.56 deg; joints [-3.922, -86.936, 146.181, -189.145, 9.398, 97.138, 179]
  MoveL 1032 to (215.09, 52.85, -4.48) mm, rotated rx -180 ry 0 rz -47.51 deg; joints [-3.922, -86.911, 146.187, -189.079, 9.476, 97.072, 179]
  MoveL 1033 to (214.85, 52.96, -4.48) mm, rotated rx 180 ry 0 rz -47.47 deg; joints [-3.922, -86.887, 146.191, -189.023, 9.543, 97.017, 179]
  MoveL 1034 to (214.61, 53.04, -4.48) mm, rotated rx -180 ry 0 rz -47.44 deg; joints [-3.922, -86.866, 146.191, -188.975, 9.6, 96.97, 179]
  MoveL 1035 to (214.37, 53.1, -4.48) mm, rotated rx 180 ry 0 rz -47.41 deg; joints [-3.921, -86.845, 146.188, -188.936, 9.648, 96.93, 179]
  MoveL 1036 to (214.36, 53.11, -4.48) mm, rotated rx -180 ry 0 rz -47.41 deg; joints [-3.921, -86.844, 146.188, -188.933, 9.651, 96.928, 179]
  MoveL 1037 to (214.12, 53.15, -4.48) mm, rotated rx -180 ry 0 rz -47.38 deg; joints [-3.921, -86.825, 146.183, -188.902, 9.689, 96.897, 179]
  MoveL 1038 to (213.88, 53.17, -4.48) mm, rotated rx -180 ry 0 rz -47.36 deg; joints [-3.921, -86.808, 146.176, -188.877, 9.72, 96.872, 179]
  MoveL 1039 to (213.4, 53.18, -4.47) mm, rotated rx -180 ry 0 rz -47.33 deg; joints [-3.92, -86.776, 146.156, -188.841, 9.763, 96.837, 179]
  MoveL 1040 to (-195.12, 53.17, -4.47) mm, rotated rx 180 ry 0 rz 63.44 deg; joints [-3.709, -54.129, 140.671, -182.204, 73.845, 90.06, 105.244]
  MoveL 1041 to (-195.28, 53.17, -4.48) mm, rotated rx 180 ry 0 rz 63.45 deg; joints [-3.709, -54.116, 140.67, -182.204, 73.856, 90.059, 105.231]
  MoveL 1042 to (-195.43, 53.16, -4.48) mm, rotated rx 180 ry 0 rz 63.46 deg; joints [-3.709, -54.103, 140.668, -182.204, 73.867, 90.059, 105.216]
  MoveL 1043 to (-195.59, 53.14, -4.47) mm, rotated rx 180 ry 0 rz 63.48 deg; joints [-3.709, -54.09, 140.666, -182.204, 73.878, 90.058, 105.199]
  MoveL 1044 to (-195.75, 53.11, -4.48) mm, rotated rx -180 ry 0 rz 63.5 deg; joints [-3.709, -54.078, 140.665, -182.204, 73.889, 90.058, 105.179]
  MoveL 1045 to (-195.92, 53.07, -4.48) mm, rotated rx 180 ry 0 rz 63.52 deg; joints [-3.709, -54.065, 140.663, -182.204, 73.9, 90.057, 105.156]
  MoveL 1046 to (-196.08, 53.02, -4.48) mm, rotated rx 180 ry 0 rz 63.55 deg; joints [-3.709, -54.052, 140.661, -182.204, 73.911, 90.057, 105.13]
  MoveL 1047 to (-196.25, 52.96, -4.48) mm, rotated rx 180 ry 0 rz 63.58 deg; joints [-3.709, -54.04, 140.66, -182.204, 73.922, 90.056, 105.102]
  MoveL 1048 to (-196.42, 52.89, -4.48) mm, rotated rx 180 ry 0 rz 63.61 deg; joints [-3.709, -54.027, 140.658, -182.204, 73.933, 90.056, 105.07]
  MoveL 1049 to (-196.56, 52.82, -4.48) mm, rotated rx -180 ry 0 rz 63.64 deg; joints [-3.71, -54.017, 140.657, -182.203, 73.942, 90.056, 105.041]
  MoveL 1050 to (-196.7, 52.74, -4.47) mm, rotated rx -180 ry 0 rz 63.67 deg; joints [-3.71, -54.007, 140.656, -182.203, 73.95, 90.055, 105.01]
  MoveL 1051 to (-196.84, 52.66, -4.48) mm, rotated rx 180 ry 0 rz 63.7 deg; joints [-3.71, -53.998, 140.654, -182.203, 73.959, 90.055, 104.977]
  MoveL 1052 to (-196.98, 52.56, -4.48) mm, rotated rx -180 ry 0 rz 63.74 deg; joints [-3.71, -53.988, 140.653, -182.203, 73.967, 90.055, 104.94]
  MoveL 1053 to (-197.12, 52.45, -4.48) mm, rotated rx -180 ry 0 rz 63.78 deg; joints [-3.71, -53.979, 140.652, -182.203, 73.975, 90.054, 104.9]
  MoveL 1054 to (-197.26, 52.33, -4.48) mm, rotated rx -180 ry 0 rz 63.82 deg; joints [-3.71, -53.97, 140.651, -182.203, 73.983, 90.054, 104.857]
  MoveL 1055 to (-197.41, 52.18, -4.48) mm, rotated rx 180 ry 0 rz 63.87 deg; joints [-3.71, -53.961, 140.649, -182.203, 73.991, 90.054, 104.806]
  MoveL 1056 to (-197.54, 52.03, -4.48) mm, rotated rx -180 ry 0 rz 63.92 deg; joints [-3.71, -53.953, 140.648, -182.203, 73.997, 90.053, 104.757]
  MoveL 1057 to (-197.7, 51.82, -4.48) mm, rotated rx 180 ry 0 rz 63.99 deg; joints [-3.71, -53.944, 140.647, -182.203, 74.005, 90.053, 104.687]
  MoveL 1058 to (-197.84, 51.6, -4.48) mm, rotated rx -180 ry 0 rz 64.06 deg; joints [-3.71, -53.938, 140.646, -182.203, 74.011, 90.053, 104.619]
  MoveL 1059 to (-197.95, 51.39, -4.48) mm, rotated rx -180 ry 0 rz 64.13 deg; joints [-3.71, -53.933, 140.646, -182.203, 74.015, 90.053, 104.553]
  MoveL 1060 to (-198.05, 51.17, -4.47) mm, rotated rx 180 ry 0 rz 64.19 deg; joints [-3.71, -53.93, 140.645, -182.203, 74.018, 90.053, 104.488]
  MoveL 1061 to (-198.13, 50.93, -4.48) mm, rotated rx 180 ry 0 rz 64.26 deg; joints [-3.71, -53.928, 140.645, -182.203, 74.02, 90.053, 104.417]
  MoveL 1062 to (-198.2, 50.69, -4.48) mm, rotated rx 180 ry 0 rz 64.33 deg; joints [-3.71, -53.927, 140.645, -182.203, 74.02, 90.053, 104.347]
  MoveL 1063 to (-198.24, 50.45, -4.48) mm, rotated rx 180 ry 0 rz 64.4 deg; joints [-3.71, -53.929, 140.645, -182.203, 74.018, 90.053, 104.278]
  MoveL 1064 to (-198.27, 50.21, -4.48) mm, rotated rx -180 ry 0 rz 64.47 deg; joints [-3.71, -53.932, 140.646, -182.203, 74.016, 90.053, 104.211]
  MoveL 1065 to (-198.27, 49.97, -4.48) mm, rotated rx -180 ry 0 rz 64.53 deg; joints [-3.71, -53.936, 140.646, -182.203, 74.012, 90.053, 104.145]
  MoveL 1066 to (-198.26, 49.73, -4.48) mm, rotated rx -180 ry 0 rz 64.6 deg; joints [-3.71, -53.943, 140.647, -182.203, 74.007, 90.053, 104.08]
  MoveL 1067 to (-198.23, 49.48, -4.48) mm, rotated rx -180 ry 0 rz 64.66 deg; joints [-3.71, -53.95, 140.648, -182.203, 74, 90.053, 104.016]
  MoveL 1068 to (-198.18, 49.24, -4.48) mm, rotated rx 180 ry 0 rz 64.73 deg; joints [-3.71, -53.959, 140.649, -182.203, 73.992, 90.054, 103.954]
  MoveL 1069 to (-198.11, 49, -4.47) mm, rotated rx 180 ry 0 rz 64.79 deg; joints [-3.71, -53.97, 140.651, -182.203, 73.983, 90.054, 103.893]
  MoveL 1070 to (-198.02, 48.76, -4.48) mm, rotated rx -180 ry 0 rz 64.85 deg; joints [-3.71, -53.983, 140.652, -182.203, 73.972, 90.054, 103.833]
  MoveL 1071 to (-197.91, 48.52, -4.47) mm, rotated rx -180 ry 0 rz 64.9 deg; joints [-3.71, -53.997, 140.654, -182.203, 73.959, 90.055, 103.775]
  MoveL 1072 to (-197.76, 48.28, -4.48) mm, rotated rx 180 ry 0 rz 64.96 deg; joints [-3.71, -54.014, 140.656, -182.203, 73.945, 90.056, 103.718]
  MoveL 1073 to (-197.66, 48.13, -4.48) mm, rotated rx -180 ry 0 rz 64.99 deg; joints [-3.709, -54.025, 140.658, -182.203, 73.935, 90.056, 103.685]
  MoveL 1074 to (-197.55, 47.98, -4.48) mm, rotated rx 180 ry 0 rz 65.03 deg; joints [-3.709, -54.038, 140.66, -182.204, 73.924, 90.056, 103.652]
  MoveL 1075 to (-197.42, 47.84, -4.48) mm, rotated rx 180 ry 0 rz 65.06 deg; joints [-3.709, -54.051, 140.661, -182.204, 73.912, 90.057, 103.62]
  MoveL 1076 to (-197.27, 47.69, -4.47) mm, rotated rx 180 ry 0 rz 65.09 deg; joints [-3.709, -54.067, 140.663, -182.204, 73.899, 90.057, 103.59]
  MoveL 1077 to (-197.03, 47.48, -4.47) mm, rotated rx 180 ry 0 rz 65.13 deg; joints [-3.709, -54.091, 140.667, -182.204, 73.877, 90.058, 103.549]
  MoveL 1078 to (-196.78, 47.31, -4.48) mm, rotated rx -180 ry 0 rz 65.16 deg; joints [-3.709, -54.115, 140.67, -182.204, 73.857, 90.059, 103.518]
  MoveL 1079 to (-196.6, 47.2, -4.48) mm, rotated rx -180 ry 0 rz 65.18 deg; joints [-3.709, -54.133, 140.672, -182.204, 73.842, 90.06, 103.501]
  Set speed (38.1 mm/s)
  MoveL 1080 to (-197.17, 46.07, -4.48) mm, rotated rx 180 ry 0 rz 65.53 deg; joints [-3.709, -54.108, 140.669, -182.204, 73.863, 90.059, 103.151]
  MoveL 1081 to (-197.73, 46.35, -4.48) mm, rotated rx 180 ry 0 rz 65.49 deg; joints [-3.709, -54.055, 140.662, -182.204, 73.909, 90.057, 103.192]
  Set speed (25.4 mm/s)
  MoveL 1082 to (-197.73, 46.35, -6.84) mm, rotated rx 180 ry 0 rz 65.49 deg; joints [-3.839, -54.053, 140.655, -182.336, 73.904, 90.065, 103.192]
  MoveL 1083 to (-197.45, 46.92, -7.47) mm, rotated rx 180 ry 0 rz 65.31 deg; joints [-3.874, -54.065, 140.655, -182.371, 73.892, 90.068, 103.366]
  Set speed (38.1 mm/s)
  MoveL 1084 to (-196.6, 47.2, -7.48) mm, rotated rx 180 ry 0 rz 65.18 deg; joints [-3.874, -54.13, 140.663, -182.372, 73.835, 90.07, 103.501]
  Set speed (76.2 mm/s)
  MoveL 1085 to (-196.42, 47.11, -7.48) mm, rotated rx -180 ry 0 rz 65.19 deg; joints [-3.874, -54.148, 140.665, -182.372, 73.82, 90.071, 103.488]
  MoveL 1086 to (-196.18, 47.01, -7.47) mm, rotated rx 180 ry 0 rz 65.2 deg; joints [-3.874, -54.17, 140.668, -182.372, 73.801, 90.072, 103.477]
  MoveL 1087 to (-195.93, 46.94, -7.48) mm, rotated rx 180 ry 0 rz 65.21 deg; joints [-3.874, -54.191, 140.671, -182.372, 73.782, 90.073, 103.472]
  MoveL 1088 to (-195.69, 46.88, -7.48) mm, rotated rx 180 ry 0 rz 65.21 deg; joints [-3.874, -54.213, 140.674, -182.373, 73.764, 90.073, 103.472]
  MoveL 1089 to (-195.45, 46.84, -7.47) mm, rotated rx 180 ry 0 rz 65.2 deg; joints [-3.874, -54.233, 140.676, -182.373, 73.746, 90.074, 103.478]
  MoveL 1090 to (-195.21, 46.83, -7.48) mm, rotated rx -180 ry 0 rz 65.19 deg; joints [-3.874, -54.254, 140.679, -182.373, 73.728, 90.075, 103.489]
  MoveL 1091 to (-194.97, 46.83, -7.47) mm, rotated rx -180 ry 0 rz 65.18 deg; joints [-3.874, -54.274, 140.682, -182.373, 73.71, 90.076, 103.505]
  MoveL 1092 to (213.41, 46.82, -7.47) mm, rotated rx -180 ry 0 rz -48.94 deg; joints [-4.081, -87.186, 145.316, -192.834, 6.952, 100.697, 179]
  MoveL 1093 to (213.89, 46.83, -7.48) mm, rotated rx -180 ry 0 rz -48.97 deg; joints [-4.082, -87.217, 145.339, -192.894, 6.918, 100.757, 179]
  MoveL 1094 to (214.13, 46.85, -7.48) mm, rotated rx 180 ry 0 rz -48.98 deg; joints [-4.083, -87.232, 145.353, -192.909, 6.91, 100.772, 179]
  MoveL 1095 to (214.37, 46.9, -7.48) mm, rotated rx 180 ry 0 rz -48.98 deg; joints [-4.083, -87.245, 145.369, -192.911, 6.911, 100.772, 179]
  MoveL 1096 to (214.63, 46.96, -7.47) mm, rotated rx 180 ry 0 rz -48.98 deg; joints [-4.084, -87.257, 145.389, -192.897, 6.921, 100.757, 179]
  MoveL 1097 to (214.88, 47.05, -7.48) mm, rotated rx 180 ry 0 rz -48.97 deg; joints [-4.085, -87.269, 145.413, -192.865, 6.941, 100.725, 179]
  MoveL 1098 to (215.01, 47.11, -7.47) mm, rotated rx -180 ry 0 rz -48.96 deg; joints [-4.085, -87.274, 145.425, -192.843, 6.956, 100.703, 179]
  MoveL 1099 to (215.14, 47.17, -7.48) mm, rotated rx -180 ry 0 rz -48.95 deg; joints [-4.086, -87.278, 145.439, -192.816, 6.973, 100.675, 179]
  MoveL 1100 to (215.26, 47.23, -7.48) mm, rotated rx -180 ry 0 rz -48.94 deg; joints [-4.086, -87.282, 145.454, -192.784, 6.993, 100.642, 179]
  MoveL 1101 to (215.39, 47.31, -7.48) mm, rotated rx -180 ry 0 rz -48.93 deg; joints [-4.087, -87.286, 145.47, -192.746, 7.017, 100.605, 179]
  MoveL 1102 to (215.62, 47.47, -7.48) mm, rotated rx 180 ry 0 rz -48.91 deg; joints [-4.088, -87.291, 145.501, -192.665, 7.069, 100.523, 179]
  MoveL 1103 to (215.84, 47.66, -7.47) mm, rotated rx -180 ry 0 rz -48.87 deg; joints [-4.089, -87.294, 145.536, -192.563, 7.134, 100.419, 179]
  MoveL 1104 to (215.98, 47.78, -7.48) mm, rotated rx -180 ry 0 rz -48.84 deg; joints [-4.09, -87.295, 145.559, -192.491, 7.181, 100.348, 179]
  MoveL 1105 to (216.1, 47.91, -7.48) mm, rotated rx -180 ry 0 rz -48.82 deg; joints [-4.09, -87.295, 145.581, -192.419, 7.229, 100.275, 179]
  MoveL 1106 to (216.2, 48.04, -7.47) mm, rotated rx -180 ry 0 rz -48.79 deg; joints [-4.091, -87.294, 145.603, -192.347, 7.277, 100.202, 179]
  MoveL 1107 to (216.3, 48.17, -7.48) mm, rotated rx -180 ry 0 rz -48.77 deg; joints [-4.092, -87.292, 145.624, -192.274, 7.326, 100.128, 179]
  MoveL 1108 to (216.39, 48.31, -7.48) mm, rotated rx 180 ry 0 rz -48.74 deg; joints [-4.092, -87.289, 145.645, -192.198, 7.378, 100.052, 179]
  MoveL 1109 to (216.47, 48.44, -7.48) mm, rotated rx -180 ry 0 rz -48.71 deg; joints [-4.093, -87.286, 145.666, -192.122, 7.431, 99.975, 179]
  MoveL 1110 to (216.54, 48.57, -7.48) mm, rotated rx -180 ry 0 rz -48.68 deg; joints [-4.093, -87.282, 145.687, -192.046, 7.484, 99.899, 179]
  MoveL 1111 to (216.6, 48.71, -7.48) mm, rotated rx -180 ry 0 rz -48.65 deg; joints [-4.094, -87.278, 145.707, -191.97, 7.538, 99.823, 179]
  MoveL 1112 to (216.66, 48.84, -7.48) mm, rotated rx -180 ry 0 rz -48.62 deg; joints [-4.095, -87.273, 145.727, -191.895, 7.592, 99.747, 179]
  MoveL 1113 to (216.71, 48.97, -7.48) mm, rotated rx -180 ry 0 rz -48.59 deg; joints [-4.095, -87.268, 145.747, -191.82, 7.647, 99.672, 179]
  MoveL 1114 to (216.75, 49.11, -7.48) mm, rotated rx -180 ry 0 rz -48.55 deg; joints [-4.096, -87.262, 145.766, -191.745, 7.703, 99.596, 179]
  MoveL 1115 to (216.79, 49.24, -7.48) mm, rotated rx -180 ry 0 rz -48.52 deg; joints [-4.096, -87.256, 145.785, -191.671, 7.759, 99.522, 179]
  MoveL 1116 to (216.84, 49.48, -7.47) mm, rotated rx -180 ry 0 rz -48.47 deg; joints [-4.097, -87.244, 145.819, -191.538, 7.861, 99.388, 179]
  MoveL 1117 to (216.87, 49.73, -7.48) mm, rotated rx 180 ry 0 rz -48.41 deg; joints [-4.098, -87.23, 145.852, -191.406, 7.965, 99.255, 179]
  MoveL 1118 to (216.88, 49.97, -7.48) mm, rotated rx -180 ry 0 rz -48.35 deg; joints [-4.099, -87.215, 145.884, -191.276, 8.07, 99.124, 179]
  MoveL 1119 to (216.87, 50.21, -7.48) mm, rotated rx -180 ry 0 rz -48.29 deg; joints [-4.1, -87.199, 145.915, -191.147, 8.176, 98.995, 179]
  MoveL 1120 to (216.85, 50.45, -7.47) mm, rotated rx 180 ry 0 rz -48.22 deg; joints [-4.1, -87.181, 145.945, -191.02, 8.285, 98.867, 179]
  MoveL 1121 to (216.8, 50.69, -7.48) mm, rotated rx 180 ry 0 rz -48.16 deg; joints [-4.101, -87.163, 145.974, -190.894, 8.394, 98.74, 179]
  MoveL 1122 to (216.74, 50.93, -7.47) mm, rotated rx 180 ry 0 rz -48.1 deg; joints [-4.102, -87.142, 146.003, -190.769, 8.506, 98.615, 179]
  MoveL 1123 to (216.65, 51.18, -7.47) mm, rotated rx 180 ry 0 rz -48.03 deg; joints [-4.102, -87.121, 146.03, -190.645, 8.619, 98.491, 179]
  MoveL 1124 to (216.58, 51.34, -7.48) mm, rotated rx 180 ry 0 rz -47.99 deg; joints [-4.103, -87.105, 146.048, -190.562, 8.697, 98.408, 179]
  MoveL 1125 to (216.5, 51.5, -7.48) mm, rotated rx 180 ry 0 rz -47.94 deg; joints [-4.103, -87.088, 146.066, -190.48, 8.775, 98.325, 179]
  MoveL 1126 to (216.41, 51.67, -7.47) mm, rotated rx -180 ry 0 rz -47.89 deg; joints [-4.103, -87.071, 146.082, -190.398, 8.855, 98.243, 179]
  MoveL 1127 to (216.3, 51.83, -7.47) mm, rotated rx -180 ry 0 rz -47.85 deg; joints [-4.104, -87.053, 146.099, -190.315, 8.936, 98.16, 179]
  MoveL 1128 to (216.2, 51.96, -7.48) mm, rotated rx -180 ry 0 rz -47.81 deg; joints [-4.104, -87.037, 146.112, -190.248, 9.004, 98.092, 179]
  MoveL 1129 to (216.09, 52.1, -7.48) mm, rotated rx -180 ry 0 rz -47.76 deg; joints [-4.104, -87.02, 146.124, -190.18, 9.073, 98.024, 179]
  MoveL 1130 to (215.96, 52.23, -7.48) mm, rotated rx -180 ry 0 rz -47.72 deg; joints [-4.104, -87.003, 146.136, -190.112, 9.143, 97.956, 179]
  MoveL 1131 to (215.82, 52.37, -7.48) mm, rotated rx -180 ry 0 rz -47.68 deg; joints [-4.105, -86.984, 146.147, -190.043, 9.215, 97.888, 179]
  MoveL 1132 to (215.58, 52.56, -7.47) mm, rotated rx -180 ry 0 rz -47.62 deg; joints [-4.105, -86.955, 146.162, -189.943, 9.321, 97.788, 179]
  MoveL 1133 to (215.34, 52.72, -7.48) mm, rotated rx -180 ry 0 rz -47.56 deg; joints [-4.105, -86.928, 146.172, -189.859, 9.412, 97.704, 179]
  MoveL 1134 to (215.09, 52.85, -7.48) mm, rotated rx -180 ry 0 rz -47.51 deg; joints [-4.105, -86.903, 146.178, -189.788, 9.49, 97.633, 179]
  MoveL 1135 to (214.85, 52.96, -7.47) mm, rotated rx -180 ry 0 rz -47.47 deg; joints [-4.105, -86.879, 146.182, -189.728, 9.557, 97.573, 179]
  MoveL 1136 to (214.61, 53.04, -7.48) mm, rotated rx 180 ry 0 rz -47.44 deg; joints [-4.104, -86.858, 146.182, -189.677, 9.614, 97.522, 179]
  MoveL 1137 to (214.37, 53.1, -7.48) mm, rotated rx 180 ry 0 rz -47.41 deg; joints [-4.104, -86.837, 146.179, -189.635, 9.662, 97.48, 179]
  MoveL 1138 to (214.36, 53.11, -7.48) mm, rotated rx 180 ry 0 rz -47.41 deg; joints [-4.104, -86.836, 146.179, -189.632, 9.665, 97.477, 179]
  MoveL 1139 to (214.12, 53.15, -7.48) mm, rotated rx -180 ry 0 rz -47.38 deg; joints [-4.104, -86.817, 146.174, -189.598, 9.703, 97.444, 179]
  MoveL 1140 to (213.88, 53.17, -7.48) mm, rotated rx 180 ry 0 rz -47.36 deg; joints [-4.103, -86.8, 146.167, -189.571, 9.733, 97.417, 179]
  MoveL 1141 to (213.4, 53.17, -7.47) mm, rotated rx 180 ry 0 rz -47.33 deg; joints [-4.103, -86.768, 146.147, -189.532, 9.776, 97.379, 179]
  MoveL 1142 to (-195.12, 53.17, -7.48) mm, rotated rx -180 ry 0 rz 63.44 deg; joints [-3.874, -54.126, 140.663, -182.372, 73.839, 90.07, 105.244]
  MoveL 1143 to (-195.28, 53.17, -7.48) mm, rotated rx -180 ry 0 rz 63.45 deg; joints [-3.874, -54.114, 140.661, -182.372, 73.85, 90.07, 105.231]
  MoveL 1144 to (-195.43, 53.16, -7.47) mm, rotated rx 180 ry 0 rz 63.46 deg; joints [-3.874, -54.101, 140.659, -182.372, 73.861, 90.069, 105.216]
  MoveL 1145 to (-195.59, 53.14, -7.48) mm, rotated rx -180 ry 0 rz 63.48 deg; joints [-3.874, -54.088, 140.658, -182.371, 73.872, 90.069, 105.199]
  MoveL 1146 to (-195.75, 53.11, -7.48) mm, rotated rx -180 ry 0 rz 63.5 deg; joints [-3.874, -54.076, 140.656, -182.371, 73.883, 90.068, 105.179]
  MoveL 1147 to (-195.92, 53.07, -7.48) mm, rotated rx 180 ry 0 rz 63.52 deg; joints [-3.874, -54.063, 140.654, -182.371, 73.894, 90.068, 105.156]
  MoveL 1148 to (-196.08, 53.02, -7.48) mm, rotated rx 180 ry 0 rz 63.55 deg; joints [-3.874, -54.05, 140.653, -182.371, 73.905, 90.067, 105.13]
  MoveL 1149 to (-196.25, 52.96, -7.48) mm, rotated rx -180 ry 0 rz 63.58 deg; joints [-3.874, -54.038, 140.651, -182.371, 73.916, 90.067, 105.102]
  MoveL 1150 to (-196.42, 52.89, -7.47) mm, rotated rx 180 ry 0 rz 63.61 deg; joints [-3.874, -54.025, 140.65, -182.371, 73.927, 90.066, 105.07]
  MoveL 1151 to (-196.56, 52.82, -7.48) mm, rotated rx -180 ry 0 rz 63.64 deg; joints [-3.874, -54.015, 140.648, -182.371, 73.935, 90.066, 105.041]
  MoveL 1152 to (-196.7, 52.74, -7.48) mm, rotated rx -180 ry 0 rz 63.67 deg; joints [-3.874, -54.005, 140.647, -182.371, 73.944, 90.066, 105.01]
  MoveL 1153 to (-196.84, 52.66, -7.48) mm, rotated rx -180 ry 0 rz 63.7 deg; joints [-3.874, -53.996, 140.646, -182.371, 73.952, 90.065, 104.977]
  MoveL 1154 to (-196.98, 52.56, -7.48) mm, rotated rx -180 ry 0 rz 63.74 deg; joints [-3.874, -53.986, 140.644, -182.371, 73.961, 90.065, 104.94]
  MoveL 1155 to (-197.12, 52.45, -7.47) mm, rotated rx -180 ry 0 rz 63.78 deg; joints [-3.874, -53.977, 140.643, -182.37, 73.969, 90.065, 104.9]
  MoveL 1156 to (-197.26, 52.33, -7.48) mm, rotated rx 180 ry 0 rz 63.82 deg; joints [-3.874, -53.968, 140.642, -182.37, 73.976, 90.064, 104.857]
  MoveL 1157 to (-197.41, 52.18, -7.48) mm, rotated rx 180 ry 0 rz 63.87 deg; joints [-3.874, -53.959, 140.641, -182.37, 73.984, 90.064, 104.806]
  MoveL 1158 to (-197.54, 52.03, -7.48) mm, rotated rx -180 ry 0 rz 63.92 deg; joints [-3.874, -53.951, 140.64, -182.37, 73.991, 90.064, 104.757]
  MoveL 1159 to (-197.7, 51.82, -7.48) mm, rotated rx -180 ry 0 rz 63.99 deg; joints [-3.874, -53.942, 140.639, -182.37, 73.999, 90.063, 104.687]
  MoveL 1160 to (-197.84, 51.6, -7.47) mm, rotated rx 180 ry 0 rz 64.06 deg; joints [-3.874, -53.936, 140.638, -182.37, 74.005, 90.063, 104.619]
  MoveL 1161 to (-197.95, 51.39, -7.48) mm, rotated rx 180 ry 0 rz 64.13 deg; joints [-3.874, -53.931, 140.637, -182.37, 74.009, 90.063, 104.553]
  MoveL 1162 to (-198.05, 51.17, -7.47) mm, rotated rx 180 ry 0 rz 64.19 deg; joints [-3.874, -53.927, 140.637, -182.37, 74.012, 90.063, 104.488]
  MoveL 1163 to (-198.13, 50.93, -7.48) mm, rotated rx -180 ry 0 rz 64.26 deg; joints [-3.874, -53.926, 140.636, -182.37, 74.013, 90.063, 104.417]
  MoveL 1164 to (-198.2, 50.69, -7.48) mm, rotated rx 180 ry 0 rz 64.33 deg; joints [-3.874, -53.925, 140.636, -182.37, 74.013, 90.063, 104.347]
  MoveL 1165 to (-198.24, 50.45, -7.47) mm, rotated rx 180 ry 0 rz 64.4 deg; joints [-3.874, -53.927, 140.637, -182.37, 74.012, 90.063, 104.278]
  MoveL 1166 to (-198.27, 50.21, -7.48) mm, rotated rx -180 ry 0 rz 64.47 deg; joints [-3.874, -53.93, 140.637, -182.37, 74.01, 90.063, 104.211]
  MoveL 1167 to (-198.27, 49.97, -7.48) mm, rotated rx 180 ry 0 rz 64.53 deg; joints [-3.874, -53.934, 140.638, -182.37, 74.006, 90.063, 104.145]
  MoveL 1168 to (-198.26, 49.73, -7.47) mm, rotated rx 180 ry 0 rz 64.6 deg; joints [-3.874, -53.94, 140.638, -182.37, 74, 90.063, 104.08]
  MoveL 1169 to (-198.23, 49.48, -7.48) mm, rotated rx -180 ry 0 rz 64.66 deg; joints [-3.874, -53.948, 140.639, -182.37, 73.994, 90.063, 104.016]
  MoveL 1170 to (-198.18, 49.24, -7.47) mm, rotated rx 180 ry 0 rz 64.73 deg; joints [-3.874, -53.957, 140.641, -182.37, 73.986, 90.064, 103.954]
  MoveL 1171 to (-198.11, 49, -7.47) mm, rotated rx 180 ry 0 rz 64.79 deg; joints [-3.874, -53.968, 140.642, -182.37, 73.977, 90.064, 103.893]
  MoveL 1172 to (-198.02, 48.76, -7.47) mm, rotated rx 180 ry 0 rz 64.85 deg; joints [-3.874, -53.98, 140.644, -182.37, 73.966, 90.065, 103.833]
  MoveL 1173 to (-197.91, 48.52, -7.47) mm, rotated rx 180 ry 0 rz 64.9 deg; joints [-3.874, -53.995, 140.646, -182.371, 73.953, 90.065, 103.775]
  MoveL 1174 to (-197.76, 48.28, -7.47) mm, rotated rx 180 ry 0 rz 64.96 deg; joints [-3.874, -54.012, 140.648, -182.371, 73.939, 90.066, 103.718]
  MoveL 1175 to (-197.66, 48.13, -7.48) mm, rotated rx 180 ry 0 rz 64.99 deg; joints [-3.874, -54.023, 140.649, -182.371, 73.929, 90.066, 103.685]
  MoveL 1176 to (-197.55, 47.98, -7.48) mm, rotated rx -180 ry 0 rz 65.03 deg; joints [-3.874, -54.036, 140.651, -182.371, 73.918, 90.067, 103.652]
  MoveL 1177 to (-197.42, 47.84, -7.48) mm, rotated rx -180 ry 0 rz 65.06 deg; joints [-3.874, -54.049, 140.653, -182.371, 73.906, 90.067, 103.62]
  MoveL 1178 to (-197.27, 47.69, -7.48) mm, rotated rx -180 ry 0 rz 65.09 deg; joints [-3.874, -54.065, 140.655, -182.371, 73.893, 90.068, 103.59]
  MoveL 1179 to (-197.03, 47.48, -7.48) mm, rotated rx -180 ry 0 rz 65.13 deg; joints [-3.874, -54.089, 140.658, -182.371, 73.871, 90.069, 103.549]
  MoveL 1180 to (-196.78, 47.31, -7.48) mm, rotated rx -180 ry 0 rz 65.16 deg; joints [-3.874, -54.113, 140.661, -182.372, 73.851, 90.07, 103.518]
  MoveL 1181 to (-196.6, 47.2, -7.48) mm, rotated rx 180 ry 0 rz 65.18 deg; joints [-3.874, -54.13, 140.663, -182.372, 73.835, 90.07, 103.501]
  Set speed (38.1 mm/s)
  MoveL 1182 to (-196.37, 46.25, -7.48) mm, rotated rx 180 ry 0 rz 65.43 deg; joints [-3.874, -54.168, 140.668, -182.372, 73.802, 90.072, 103.254]
  MoveL 1183 to (-198.16, 43.86, -7.48) mm, rotated rx 180 ry 0 rz 66.2 deg; joints [-3.874, -54.064, 140.655, -182.371, 73.893, 90.068, 102.482]
  MoveL 1184 to (-198.54, 43.36, -6.84) mm, rotated rx 180 ry 0 rz 66.36 deg; joints [-3.839, -54.042, 140.654, -182.336, 73.914, 90.065, 102.318]
  Set speed (100.0 mm/s)
  MoveL 1185 to (-198.54, 43.36, 24.52) mm, rotated rx 180 ry 0 rz 66.36 deg; joints [-2.115, -54.055, 140.712, -180.585, 73.956, 89.958, 102.318]
  MoveL 1186 to (-195.3, 420.76, 24.52) mm, rotated rx -180 ry 0 rz 13.58 deg; joints [-2.138, -31.914, 134.438, -180.584, 89.823, 89.794, 155.102]
  MoveL 1187 to (-195.3, 420.76, 3.11) mm, rotated rx 180 ry 0 rz 13.58 deg; joints [-3.322, -31.918, 134.408, -181.739, 89.784, 89.538, 155.102]
  Set speed (25.4 mm/s)
  MoveL 1188 to (-195.3, 420.76, -0.84) mm, rotated rx -180 ry 0 rz 13.58 deg; joints [-3.541, -31.919, 134.4, -181.953, 89.773, 89.491, 155.102]
  MoveL 1189 to (-195.48, 421.37, -1.47) mm, rotated rx -180 ry 0 rz 13.57 deg; joints [-3.576, -31.868, 134.376, -181.987, 89.8, 89.482, 155.113]
  Set speed (38.1 mm/s)
  MoveL 1190 to (-195.58, 421.7, -1.47) mm, rotated rx 180 ry 0 rz 13.56 deg; joints [-3.576, -31.839, 134.363, -181.987, 89.816, 89.482, 155.119]
  MoveL 1191 to (-194.97, 422.52, -1.47) mm, rotated rx -180 ry 0 rz 13.45 deg; joints [-3.576, -31.8, 134.346, -181.987, 89.838, 89.481, 155.229]
  Set speed (76.2 mm/s)
  MoveL 1192 to (213.41, 422.52, -1.48) mm, rotated rx -180 ry 0 rz -38.12 deg; joints [-3.904, -49.126, 150.459, -182.018, 60.827, 89.38, 179]
  MoveL 1193 to (213.89, 422.53, -1.48) mm, rotated rx -180 ry 0 rz -38.17 deg; joints [-3.904, -49.151, 150.485, -182.018, 60.776, 89.38, 179]
  MoveL 1194 to (214.13, 422.55, -1.47) mm, rotated rx -180 ry 0 rz -38.19 deg; joints [-3.905, -49.161, 150.497, -182.018, 60.754, 89.379, 179]
  MoveL 1195 to (214.37, 422.59, -1.48) mm, rotated rx 180 ry 0 rz -38.22 deg; joints [-3.905, -49.168, 150.509, -182.018, 60.735, 89.379, 179]
  MoveL 1196 to (214.61, 422.65, -1.48) mm, rotated rx 180 ry 0 rz -38.24 deg; joints [-3.906, -49.173, 150.521, -182.018, 60.72, 89.378, 179]
  MoveL 1197 to (214.85, 422.74, -1.48) mm, rotated rx -180 ry 0 rz -38.26 deg; joints [-3.906, -49.175, 150.533, -182.018, 60.709, 89.378, 179]
  MoveL 1198 to (215.09, 422.84, -1.47) mm, rotated rx 180 ry 0 rz -38.28 deg; joints [-3.906, -49.173, 150.544, -182.018, 60.701, 89.377, 179]
  MoveL 1199 to (215.34, 422.97, -1.48) mm, rotated rx -180 ry 0 rz -38.3 deg; joints [-3.907, -49.169, 150.555, -182.018, 60.698, 89.376, 179]
  MoveL 1200 to (215.58, 423.13, -1.47) mm, rotated rx 180 ry 0 rz -38.32 deg; joints [-3.907, -49.161, 150.566, -182.018, 60.699, 89.375, 179]
  MoveL 1201 to (215.82, 423.33, -1.48) mm, rotated rx 180 ry 0 rz -38.33 deg; joints [-3.908, -49.148, 150.576, -182.017, 60.707, 89.374, 179]
  MoveL 1202 to (215.96, 423.46, -1.47) mm, rotated rx 180 ry 0 rz -38.34 deg; joints [-3.908, -49.137, 150.582, -182.017, 60.716, 89.373, 179]
  MoveL 1203 to (216.09, 423.6, -1.48) mm, rotated rx -180 ry 0 rz -38.35 deg; joints [-3.909, -49.126, 150.587, -182.017, 60.725, 89.372, 179]
  MoveL 1204 to (216.2, 423.73, -1.47) mm, rotated rx 180 ry 0 rz -38.35 deg; joints [-3.909, -49.114, 150.591, -182.017, 60.737, 89.372, 179]
  MoveL 1205 to (216.3, 423.87, -1.48) mm, rotated rx -180 ry 0 rz -38.36 deg; joints [-3.909, -49.102, 150.595, -182.017, 60.75, 89.371, 179]
  MoveL 1206 to (216.39, 424.01, -1.48) mm, rotated rx -180 ry 0 rz -38.36 deg; joints [-3.909, -49.088, 150.598, -182.017, 60.764, 89.37, 179]
  MoveL 1207 to (216.47, 424.15, -1.48) mm, rotated rx -180 ry 0 rz -38.36 deg; joints [-3.91, -49.074, 150.6, -182.017, 60.779, 89.37, 179]
  MoveL 1208 to (216.6, 424.39, -1.47) mm, rotated rx 180 ry 0 rz -38.36 deg; joints [-3.91, -49.049, 150.604, -182.016, 60.808, 89.368, 179]
  MoveL 1209 to (216.69, 424.63, -1.47) mm, rotated rx 180 ry 0 rz -38.36 deg; joints [-3.91, -49.022, 150.606, -182.016, 60.839, 89.367, 179]
  MoveL 1210 to (216.77, 424.87, -1.48) mm, rotated rx -180 ry 0 rz -38.35 deg; joints [-3.911, -48.994, 150.606, -182.016, 60.873, 89.366, 179]
  MoveL 1211 to (216.82, 425.11, -1.47) mm, rotated rx 180 ry 0 rz -38.34 deg; joints [-3.911, -48.965, 150.606, -182.016, 60.909, 89.365, 179]
  MoveL 1212 to (216.86, 425.35, -1.47) mm, rotated rx 180 ry 0 rz -38.33 deg; joints [-3.911, -48.935, 150.605, -182.015, 60.947, 89.364, 179]
  MoveL 1213 to (216.88, 425.59, -1.48) mm, rotated rx -180 ry 0 rz -38.32 deg; joints [-3.911, -48.904, 150.602, -182.015, 60.987, 89.362, 179]
  MoveL 1214 to (216.88, 425.84, -1.48) mm, rotated rx -180 ry 0 rz -38.31 deg; joints [-3.912, -48.872, 150.599, -182.015, 61.029, 89.361, 179]
  MoveL 1215 to (216.87, 426.08, -1.48) mm, rotated rx 180 ry 0 rz -38.3 deg; joints [-3.912, -48.84, 150.596, -182.015, 61.071, 89.36, 179]
  MoveL 1216 to (216.85, 426.28, -1.48) mm, rotated rx -180 ry 0 rz -38.28 deg; joints [-3.912, -48.812, 150.592, -182.015, 61.108, 89.359, 179]
  MoveL 1217 to (216.82, 426.49, -1.47) mm, rotated rx 180 ry 0 rz -38.27 deg; joints [-3.912, -48.783, 150.587, -182.014, 61.147, 89.358, 179]
  MoveL 1218 to (216.77, 426.69, -1.48) mm, rotated rx -180 ry 0 rz -38.25 deg; joints [-3.912, -48.754, 150.582, -182.014, 61.187, 89.357, 179]
  MoveL 1219 to (216.71, 426.89, -1.48) mm, rotated rx -180 ry 0 rz -38.24 deg; joints [-3.912, -48.724, 150.576, -182.014, 61.229, 89.357, 179]
  MoveL 1220 to (216.64, 427.1, -1.48) mm, rotated rx -180 ry 0 rz -38.22 deg; joints [-3.912, -48.693, 150.569, -182.014, 61.272, 89.356, 179]
  MoveL 1221 to (216.54, 427.3, -1.48) mm, rotated rx -180 ry 0 rz -38.19 deg; joints [-3.912, -48.661, 150.561, -182.014, 61.317, 89.355, 179]
  MoveL 1222 to (216.43, 427.51, -1.48) mm, rotated rx -180 ry 0 rz -38.17 deg; joints [-3.912, -48.628, 150.552, -182.013, 61.364, 89.354, 179]
  MoveL 1223 to (216.3, 427.71, -1.47) mm, rotated rx 180 ry 0 rz -38.15 deg; joints [-3.912, -48.595, 150.542, -182.013, 61.413, 89.353, 179]
  MoveL 1224 to (216.19, 427.86, -1.48) mm, rotated rx -180 ry 0 rz -38.13 deg; joints [-3.912, -48.569, 150.534, -182.013, 61.45, 89.353, 179]
  MoveL 1225 to (216.06, 428.01, -1.48) mm, rotated rx -180 ry 0 rz -38.1 deg; joints [-3.912, -48.542, 150.525, -182.013, 61.49, 89.352, 179]
  MoveL 1226 to (215.85, 428.22, -1.48) mm, rotated rx -180 ry 0 rz -38.07 deg; joints [-3.912, -48.504, 150.511, -182.013, 61.548, 89.351, 179]
  MoveL 1227 to (215.64, 428.4, -1.48) mm, rotated rx -180 ry 0 rz -38.04 deg; joints [-3.912, -48.469, 150.497, -182.013, 61.601, 89.351, 179]
  MoveL 1228 to (215.43, 428.55, -1.47) mm, rotated rx 180 ry 0 rz -38.01 deg; joints [-3.911, -48.439, 150.484, -182.013, 61.648, 89.35, 179]
  MoveL 1229 to (215.21, 428.67, -1.48) mm, rotated rx -180 ry 0 rz -37.98 deg; joints [-3.911, -48.411, 150.471, -182.012, 61.692, 89.35, 179]
  MoveL 1230 to (215, 428.78, -1.48) mm, rotated rx -180 ry 0 rz -37.95 deg; joints [-3.911, -48.387, 150.458, -182.012, 61.732, 89.35, 179]
  MoveL 1231 to (214.79, 428.86, -1.47) mm, rotated rx 180 ry 0 rz -37.92 deg; joints [-3.911, -48.364, 150.445, -182.012, 61.768, 89.35, 179]
  MoveL 1232 to (214.58, 428.93, -1.48) mm, rotated rx -180 ry 0 rz -37.9 deg; joints [-3.91, -48.344, 150.433, -182.012, 61.802, 89.35, 179]
  MoveL 1233 to (214.37, 428.98, -1.48) mm, rotated rx -180 ry 0 rz -37.87 deg; joints [-3.91, -48.327, 150.421, -182.012, 61.833, 89.35, 179]
  MoveL 1234 to (214.13, 429.03, -1.47) mm, rotated rx 180 ry 0 rz -37.84 deg; joints [-3.91, -48.308, 150.407, -182.012, 61.866, 89.35, 179]
  MoveL 1235 to (213.89, 429.05, -1.47) mm, rotated rx 180 ry 0 rz -37.82 deg; joints [-3.909, -48.293, 150.394, -182.012, 61.895, 89.35, 179]
  MoveL 1236 to (213.41, 429.06, -1.47) mm, rotated rx -180 ry 0 rz -37.77 deg; joints [-3.908, -48.267, 150.368, -182.012, 61.947, 89.35, 179]
  MoveL 1237 to (-194.97, 429.06, -1.48) mm, rotated rx 180 ry 0 rz 13.12 deg; joints [-3.577, -31.316, 134.13, -181.988, 90.106, 89.471, 155.562]
  MoveL 1238 to (-195.21, 429.05, -1.48) mm, rotated rx 180 ry 0 rz 13.14 deg; joints [-3.577, -31.308, 134.127, -181.988, 90.111, 89.471, 155.535]
  MoveL 1239 to (-195.45, 429.04, -1.48) mm, rotated rx -180 ry 0 rz 13.17 deg; joints [-3.577, -31.301, 134.124, -181.988, 90.115, 89.471, 155.508]
  MoveL 1240 to (-195.69, 429, -1.48) mm, rotated rx 180 ry 0 rz 13.2 deg; joints [-3.577, -31.295, 134.121, -181.988, 90.118, 89.471, 155.479]
  MoveL 1241 to (-195.93, 428.94, -1.48) mm, rotated rx -180 ry 0 rz 13.23 deg; joints [-3.577, -31.291, 134.119, -181.988, 90.12, 89.471, 155.45]
  MoveL 1242 to (-196.18, 428.87, -1.48) mm, rotated rx 180 ry 0 rz 13.26 deg; joints [-3.577, -31.289, 134.118, -181.988, 90.121, 89.471, 155.419]
  MoveL 1243 to (-196.42, 428.77, -1.48) mm, rotated rx 180 ry 0 rz 13.29 deg; joints [-3.577, -31.288, 134.118, -181.988, 90.122, 89.471, 155.388]
  MoveL 1244 to (-196.55, 428.71, -1.48) mm, rotated rx 180 ry 0 rz 13.31 deg; joints [-3.577, -31.288, 134.118, -181.988, 90.122, 89.471, 155.37]
  MoveL 1245 to (-196.68, 428.64, -1.47) mm, rotated rx 180 ry 0 rz 13.33 deg; joints [-3.577, -31.289, 134.118, -181.988, 90.121, 89.471, 155.352]
  MoveL 1246 to (-196.81, 428.56, -1.48) mm, rotated rx -180 ry 0 rz 13.35 deg; joints [-3.577, -31.29, 134.119, -181.988, 90.12, 89.471, 155.334]
  MoveL 1247 to (-196.93, 428.47, -1.48) mm, rotated rx 180 ry 0 rz 13.36 deg; joints [-3.577, -31.292, 134.12, -181.988, 90.119, 89.471, 155.315]
  MoveL 1248 to (-197.06, 428.37, -1.48) mm, rotated rx 180 ry 0 rz 13.38 deg; joints [-3.577, -31.295, 134.121, -181.988, 90.118, 89.471, 155.296]
  MoveL 1249 to (-197.19, 428.27, -1.48) mm, rotated rx 180 ry 0 rz 13.4 deg; joints [-3.577, -31.299, 134.123, -181.988, 90.116, 89.471, 155.276]
  MoveL 1250 to (-197.32, 428.15, -1.48) mm, rotated rx 180 ry 0 rz 13.42 deg; joints [-3.577, -31.303, 134.125, -181.988, 90.113, 89.471, 155.256]
  MoveL 1251 to (-197.45, 428.01, -1.47) mm, rotated rx 180 ry 0 rz 13.44 deg; joints [-3.577, -31.309, 134.127, -181.988, 90.11, 89.471, 155.235]
  MoveL 1252 to (-197.65, 427.77, -1.48) mm, rotated rx 180 ry 0 rz 13.48 deg; joints [-3.577, -31.32, 134.132, -181.988, 90.104, 89.472, 155.201]
  MoveL 1253 to (-197.81, 427.53, -1.48) mm, rotated rx 180 ry 0 rz 13.51 deg; joints [-3.577, -31.332, 134.138, -181.988, 90.097, 89.472, 155.171]
  MoveL 1254 to (-197.94, 427.29, -1.48) mm, rotated rx 180 ry 0 rz 13.54 deg; joints [-3.577, -31.346, 134.144, -181.988, 90.09, 89.472, 155.144]
  MoveL 1255 to (-198.05, 427.04, -1.48) mm, rotated rx -180 ry 0 rz 13.56 deg; joints [-3.577, -31.36, 134.15, -181.988, 90.082, 89.472, 155.119]
  MoveL 1256 to (-198.14, 426.8, -1.47) mm, rotated rx 180 ry 0 rz 13.58 deg; joints [-3.577, -31.375, 134.157, -181.988, 90.074, 89.473, 155.098]
  MoveL 1257 to (-198.2, 426.56, -1.48) mm, rotated rx 180 ry 0 rz 13.6 deg; joints [-3.576, -31.39, 134.164, -181.988, 90.065, 89.473, 155.078]
  MoveL 1258 to (-198.24, 426.32, -1.48) mm, rotated rx 180 ry 0 rz 13.62 deg; joints [-3.576, -31.407, 134.171, -181.988, 90.056, 89.473, 155.061]
  MoveL 1259 to (-198.27, 426.08, -1.47) mm, rotated rx 180 ry 0 rz 13.63 deg; joints [-3.576, -31.424, 134.179, -181.988, 90.047, 89.474, 155.046]
  MoveL 1260 to (-198.27, 425.84, -1.48) mm, rotated rx 180 ry 0 rz 13.65 deg; joints [-3.576, -31.441, 134.187, -181.988, 90.037, 89.474, 155.033]
  MoveL 1261 to (-198.27, 425.59, -1.48) mm, rotated rx 180 ry 0 rz 13.66 deg; joints [-3.576, -31.459, 134.194, -181.988, 90.027, 89.474, 155.021]
  MoveL 1262 to (-198.25, 425.35, -1.48) mm, rotated rx -180 ry 0 rz 13.67 deg; joints [-3.576, -31.478, 134.203, -181.988, 90.017, 89.475, 155.01]
  MoveL 1263 to (-198.22, 425.11, -1.47) mm, rotated rx -180 ry 0 rz 13.68 deg; joints [-3.576, -31.497, 134.211, -181.988, 90.006, 89.475, 155.002]
  MoveL 1264 to (-198.16, 424.87, -1.48) mm, rotated rx 180 ry 0 rz 13.68 deg; joints [-3.576, -31.516, 134.22, -181.987, 89.996, 89.475, 154.995]
  MoveL 1265 to (-198.09, 424.63, -1.48) mm, rotated rx 180 ry 0 rz 13.69 deg; joints [-3.576, -31.537, 134.229, -181.987, 89.984, 89.476, 154.991]
  MoveL 1266 to (-197.99, 424.39, -1.48) mm, rotated rx 180 ry 0 rz 13.69 deg; joints [-3.576, -31.558, 134.239, -181.987, 89.972, 89.476, 154.989]
  MoveL 1267 to (-197.87, 424.15, -1.48) mm, rotated rx 180 ry 0 rz 13.69 deg; joints [-3.576, -31.58, 134.248, -181.987, 89.96, 89.477, 154.991]
  MoveL 1268 to (-197.73, 423.93, -1.48) mm, rotated rx -180 ry 0 rz 13.69 deg; joints [-3.576, -31.601, 134.258, -181.987, 89.949, 89.477, 154.994]
  MoveL 1269 to (-197.57, 423.71, -1.48) mm, rotated rx -180 ry 0 rz 13.68 deg; joints [-3.576, -31.623, 134.267, -181.987, 89.937, 89.477, 155.001]
  MoveL 1270 to (-197.38, 423.49, -1.47) mm, rotated rx -180 ry 0 rz 13.67 deg; joints [-3.576, -31.646, 134.277, -181.987, 89.924, 89.478, 155.011]
  MoveL 1271 to (-197.14, 423.27, -1.48) mm, rotated rx 180 ry 0 rz 13.65 deg; joints [-3.576, -31.67, 134.288, -181.987, 89.91, 89.478, 155.026]
  MoveL 1272 to (-196.96, 423.13, -1.47) mm, rotated rx 180 ry 0 rz 13.64 deg; joints [-3.576, -31.687, 134.296, -181.987, 89.901, 89.479, 155.038]
  MoveL 1273 to (-196.78, 423, -1.48) mm, rotated rx -180 ry 0 rz 13.63 deg; joints [-3.576, -31.702, 134.302, -181.987, 89.892, 89.479, 155.052]
  MoveL 1274 to (-196.6, 422.9, -1.48) mm, rotated rx 180 ry 0 rz 13.61 deg; joints [-3.576, -31.716, 134.309, -181.987, 89.885, 89.479, 155.067]
  MoveL 1275 to (-196.42, 422.81, -1.48) mm, rotated rx -180 ry 0 rz 13.6 deg; joints [-3.576, -31.729, 134.314, -181.987, 89.877, 89.48, 155.083]
  MoveL 1276 to (-196.18, 422.71, -1.47) mm, rotated rx 180 ry 0 rz 13.58 deg; joints [-3.576, -31.744, 134.321, -181.987, 89.869, 89.48, 155.104]
  MoveL 1277 to (-195.93, 422.63, -1.48) mm, rotated rx -180 ry 0 rz 13.55 deg; joints [-3.576, -31.758, 134.327, -181.987, 89.861, 89.48, 155.127]
  MoveL 1278 to (-195.69, 422.58, -1.47) mm, rotated rx 180 ry 0 rz 13.53 deg; joints [-3.576, -31.771, 134.333, -181.987, 89.854, 89.48, 155.151]
